LIN {X 0,Y 469.343,Z 366.999,A -85,B 0,C 180,E1 -7684.11,E2 -7684.11} C_VEL
LIN {X 0,Y 469.709,Z 359.682,A -85,B 0,C 180,E1 -7686.102,E2 -7686.102} C_VEL
LIN {X 0,Y 468.782,Z 353.417,A -85,B 0,C 180,E1 -7687.929,E2 -7687.929} C_VEL
LIN {X 0,Y 467.594,Z 347.243,A -85,B 0,C 180,E1 -7689.819,E2 -7689.819} C_VEL
LIN {X 0,Y 467.591,Z 347.243,A -85,B 0,C 180,E1 -7692.567,E2 -7692.567} C_VEL
LIN {X 0,Y 467.575,Z 347.246,A -85,B 0,C 180,E1 -7695.054,E2 -7695.054} C_VEL
LIN {X 0,Y 467.593,Z 347.241,A -85,B 0,C 180,E1 -7697.44,E2 -7697.44} C_VEL
LIN {X 0,Y 467.587,Z 347.243,A -85,B 0,C 180,E1 -7700.856,E2 -7700.856} C_VEL
LIN {X 0,Y 467.564,Z 347.245,A -85,B 0,C 180,E1 -7704.261,E2 -7704.261} C_VEL
LIN {X 0,Y 467.587,Z 347.242,A -85,B 0,C 180,E1 -7707.321,E2 -7707.321} C_VEL
LIN {X 0,Y 467.575,Z 347.245,A -85,B 0,C 180,E1 -7710.668,E2 -7710.668} C_VEL
LIN {X 0,Y 467.622,Z 347.237,A -85,B 0,C 180,E1 -7713.2,E2 -7713.2} C_VEL
LIN {X 0,Y 467.598,Z 347.242,A -85,B 0,C 180,E1 -7716.468,E2 -7716.468} C_VEL
LIN {X 0,Y 467.628,Z 347.236,A -85,B 0,C 180,E1 -7719.777,E2 -7719.777} C_VEL
LIN {X 0,Y 467.605,Z 347.24,A -85,B 0,C 180,E1 -7722.507,E2 -7722.507} C_VEL
LIN {X 0,Y 467.612,Z 347.238,A -85,B 0,C 180,E1 -7725.197,E2 -7725.197} C_VEL
LIN {X 0,Y 467.662,Z 347.233,A -85,B 0,C 180,E1 -7727.855,E2 -7727.855} C_VEL
LIN {X 0,Y 467.686,Z 347.227,A -85,B 0,C 180,E1 -7731.357,E2 -7731.357} C_VEL
LIN {X 0,Y 467.75,Z 347.221,A -85,B 0,C 180,E1 -7733.963,E2 -7733.963} C_VEL
LIN {X 0,Y 467.864,Z 347.206,A -85,B 0,C 180,E1 -7737.417,E2 -7737.417} C_VEL
LIN {X 0,Y 467.889,Z 347.206,A -85,B 0,C 180,E1 -7740,E2 -7740} C_VEL
LIN {X 0,Y 467.865,Z 347.207,A -85,B 0,C 180,E1 -7742.583,E2 -7742.583} C_VEL
LIN {X 0,Y 467.749,Z 347.222,A -85,B 0,C 180,E1 -7746.038,E2 -7746.038} C_VEL
LIN {X 0,Y 467.688,Z 347.229,A -85,B 0,C 180,E1 -7748.643,E2 -7748.643} C_VEL
LIN {X 0,Y 467.663,Z 347.235,A -85,B 0,C 180,E1 -7752.146,E2 -7752.146} C_VEL
LIN {X 0,Y 467.646,Z 347.236,A -85,B 0,C 180,E1 -7755.695,E2 -7755.695} C_VEL
LIN {X 0,Y 467.624,Z 347.236,A -85,B 0,C 180,E1 -7758.765,E2 -7758.765} C_VEL
LIN {X 0,Y 467.587,Z 347.242,A -85,B 0,C 180,E1 -7761.268,E2 -7761.268} C_VEL
LIN {X 0,Y 467.58,Z 347.243,A -85,B 0,C 180,E1 -7763.943,E2 -7763.943} C_VEL
LIN {X 0,Y 467.623,Z 347.236,A -85,B 0,C 180,E1 -7766.8,E2 -7766.8} C_VEL
LIN {X 0,Y 467.56,Z 347.246,A -85,B 0,C 180,E1 -7769.738,E2 -7769.738} C_VEL
LIN {X 0,Y 467.59,Z 347.241,A -85,B 0,C 180,E1 -7772.758,E2 -7772.758} C_VEL
LIN {X 0,Y 467.56,Z 347.245,A -85,B 0,C 180,E1 -7775.89,E2 -7775.89} C_VEL
LIN {X 0,Y 467.589,Z 347.242,A -85,B 0,C 180,E1 -7779.145,E2 -7779.145} C_VEL
LIN {X 0,Y 467.593,Z 347.24,A -85,B 0,C 180,E1 -7782.567,E2 -7782.567} C_VEL
LIN {X 0,Y 467.577,Z 347.244,A -85,B 0,C 180,E1 -7785.053,E2 -7785.053} C_VEL
LIN {X 0,Y 467.595,Z 347.241,A -85,B 0,C 180,E1 -7787.44,E2 -7787.44} C_VEL
LIN {X 0,Y 467.588,Z 347.242,A -85,B 0,C 180,E1 -7790.855,E2 -7790.855} C_VEL
LIN {X 0,Y 467.564,Z 347.243,A -85,B 0,C 180,E1 -7794.261,E2 -7794.261} C_VEL
LIN {X 0,Y 467.589,Z 347.242,A -85,B 0,C 180,E1 -7797.321,E2 -7797.321} C_VEL
LIN {X 0,Y 467.576,Z 347.245,A -85,B 0,C 180,E1 -7800.667,E2 -7800.667} C_VEL
LIN {X 0,Y 467.623,Z 347.238,A -85,B 0,C 180,E1 -7803.199,E2 -7803.199} C_VEL
LIN {X 0,Y 467.599,Z 347.241,A -85,B 0,C 180,E1 -7806.468,E2 -7806.468} C_VEL
LIN {X 0,Y 467.63,Z 347.235,A -85,B 0,C 180,E1 -7809.777,E2 -7809.777} C_VEL
LIN {X 0,Y 467.614,Z 347.239,A -85,B 0,C 180,E1 -7812.506,E2 -7812.506} C_VEL
LIN {X 0,Y 467.604,Z 347.238,A -85,B 0,C 180,E1 -7815.421,E2 -7815.421} C_VEL
LIN {X 0,Y 466.933,Z 347.324,A -85,B 0,C 180,E1 -7816.14,E2 -7816.14} C_VEL
LIN {X 0,Y 464.09,Z 347.677,A -85,B 0,C 180,E1 -7817.309,E2 -7817.309} C_VEL
LIN {X 0,Y 461.692,Z 347.976,A -85,B 0,C 180,E1 -7818.251,E2 -7818.251} C_VEL
LIN {X 0,Y 460.666,Z 348.105,A -85,B 0,C 180,E1 -7818.978,E2 -7818.978} C_VEL
LIN {X 0,Y 460.584,Z 348.115,A -85,B 0,C 180,E1 -7819.225,E2 -7819.225} C_VEL
LIN {X 0,Y 460.675,Z 348.104,A -85,B 0,C 180,E1 -7822.587,E2 -7822.587} C_VEL
LIN {X 0,Y 460.674,Z 348.304,A -85,B 0,C 180,E1 -7822.926,E2 -7822.926} C_VEL
LIN {X 0,Y 463.587,Z 358.571,A -85,B 0,C 180,E1 -7823.471,E2 -7823.471} C_VEL
LIN {X 0,Y 463.267,Z 370.178,A -85,B 0,C 180,E1 -7824.122,E2 -7824.122} C_VEL
LIN {X 0,Y 462.868,Z 380.748,A -85,B 0,C 180,E1 -7824.882,E2 -7824.882} C_VEL
LIN {X 0,Y 462.353,Z 391.565,A -85,B 0,C 180,E1 -7825.859,E2 -7825.859} C_VEL
LIN {X 0,Y 461.872,Z 401.21,A -85,B 0,C 180,E1 -7826.947,E2 -7826.947} C_VEL
LIN {X 0,Y 461.389,Z 410.564,A -85,B 0,C 180,E1 -7828.254,E2 -7828.254} C_VEL
LIN {X 0,Y 460.955,Z 418.019,A -85,B 0,C 180,E1 -7829.563,E2 -7829.563} C_VEL
LIN {X 0,Y 460.616,Z 424.017,A -85,B 0,C 180,E1 -7830.874,E2 -7830.874} C_VEL
LIN {X 0,Y 460.424,Z 428.772,A -85,B 0,C 180,E1 -7832.186,E2 -7832.186} C_VEL
LIN {X 0,Y 460.216,Z 432.455,A -85,B 0,C 180,E1 -7833.501,E2 -7833.501} C_VEL
LIN {X 0,Y 460.141,Z 434.354,A -85,B 0,C 180,E1 -7834.379,E2 -7834.379} C_VEL
LIN {X 0,Y 460.106,Z 435.844,A -85,B 0,C 180,E1 -7835.258,E2 -7835.258} C_VEL
LIN {X 0,Y 460.098,Z 437.555,A -85,B 0,C 180,E1 -7837.018,E2 -7837.018} C_VEL
LIN {X 0,Y 460.068,Z 437.759,A -85,B 0,C 180,E1 -7838.786,E2 -7838.786} C_VEL
LIN {X 0,Y 460.068,Z 436.331,A -85,B 0,C 180,E1 -7840.562,E2 -7840.562} C_VEL
LIN {X 0,Y 460.31,Z 433.443,A -85,B 0,C 180,E1 -7842.27,E2 -7842.27} C_VEL
LIN {X 0,Y 460.472,Z 429.812,A -85,B 0,C 180,E1 -7843.684,E2 -7843.684} C_VEL
LIN {X 0,Y 460.719,Z 425.206,A -85,B 0,C 180,E1 -7845.029,E2 -7845.029} C_VEL
LIN {X 0,Y 461.101,Z 418.242,A -85,B 0,C 180,E1 -7846.596,E2 -7846.596} C_VEL
LIN {X 0,Y 461.515,Z 410.521,A -85,B 0,C 180,E1 -7847.96,E2 -7847.96} C_VEL
LIN {X 0,Y 462.079,Z 401.988,A -85,B 0,C 180,E1 -7849.162,E2 -7849.162} C_VEL
LIN {X 0,Y 462.433,Z 392.799,A -85,B 0,C 180,E1 -7850.227,E2 -7850.227} C_VEL
LIN {X 0,Y 462.997,Z 381.824,A -85,B 0,C 180,E1 -7851.247,E2 -7851.247} C_VEL
LIN {X 0,Y 463.474,Z 370.955,A -85,B 0,C 180,E1 -7852.042,E2 -7852.042} C_VEL
LIN {X 0,Y 463.827,Z 358.885,A -85,B 0,C 180,E1 -7852.728,E2 -7852.728} C_VEL
LIN {X 0,Y 460.571,Z 348.116,A -85,B 0,C 180,E1 -7853.333,E2 -7853.333} C_VEL
LIN {X 0,Y 460.566,Z 348.118,A -85,B 0,C 180,E1 -7856.264,E2 -7856.264} C_VEL
LIN {X 0,Y 460.542,Z 348.122,A -85,B 0,C 180,E1 -7859.23,E2 -7859.23} C_VEL
LIN {X 0,Y 460.533,Z 348.125,A -85,B 0,C 180,E1 -7862.283,E2 -7862.283} C_VEL
LIN {X 0,Y 460.511,Z 348.127,A -85,B 0,C 180,E1 -7865.445,E2 -7865.445} C_VEL
LIN {X 0,Y 460.545,Z 348.12,A -85,B 0,C 180,E1 -7868.897,E2 -7868.897} C_VEL
LIN {X 0,Y 460.524,Z 348.121,A -85,B 0,C 180,E1 -7872.18,E2 -7872.18} C_VEL
LIN {X 0,Y 460.517,Z 348.125,A -85,B 0,C 180,E1 -7875.411,E2 -7875.411} C_VEL
LIN {X 0,Y 460.535,Z 348.123,A -85,B 0,C 180,E1 -7878.396,E2 -7878.396} C_VEL
LIN {X 0,Y 460.546,Z 348.12,A -85,B 0,C 180,E1 -7881.268,E2 -7881.268} C_VEL
LIN {X 0,Y 460.513,Z 348.124,A -85,B 0,C 180,E1 -7884.554,E2 -7884.554} C_VEL
LIN {X 0,Y 460.531,Z 348.116,A -85,B 0,C 180,E1 -7887.715,E2 -7887.715} C_VEL
LIN {X 0,Y 460.546,Z 348.106,A -85,B 0,C 180,E1 -7890.769,E2 -7890.769} C_VEL
LIN {X 0,Y 460.566,Z 348.116,A -85,B 0,C 180,E1 -7893.735,E2 -7893.735} C_VEL
LIN {X 0,Y 460.544,Z 348.114,A -85,B 0,C 180,E1 -7896.623,E2 -7896.623} C_VEL
LIN {X 0,Y 460.55,Z 348.12,A -85,B 0,C 180,E1 -7899.452,E2 -7899.452} C_VEL
LIN {X 0,Y 460.557,Z 348.113,A -85,B 0,C 180,E1 -7902.23,E2 -7902.23} C_VEL
LIN {X 0,Y 460.565,Z 348.117,A -85,B 0,C 180,E1 -7904.965,E2 -7904.965} C_VEL
LIN {X 0,Y 460.628,Z 348.109,A -85,B 0,C 180,E1 -7907.666,E2 -7907.666} C_VEL
LIN {X 0,Y 460.627,Z 348.11,A -85,B 0,C 180,E1 -7911.224,E2 -7911.224} C_VEL
LIN {X 0,Y 460.707,Z 348.094,A -85,B 0,C 180,E1 -7913.87,E2 -7913.87} C_VEL
LIN {X 0,Y 460.823,Z 348.086,A -85,B 0,C 180,E1 -7917.377,E2 -7917.377} C_VEL
LIN {X 0,Y 460.851,Z 348.076,A -85,B 0,C 180,E1 -7920,E2 -7920} C_VEL
LIN {X 0,Y 460.822,Z 348.085,A -85,B 0,C 180,E1 -7922.622,E2 -7922.622} C_VEL
LIN {X 0,Y 460.707,Z 348.097,A -85,B 0,C 180,E1 -7926.13,E2 -7926.13} C_VEL
LIN {X 0,Y 460.625,Z 348.108,A -85,B 0,C 180,E1 -7928.776,E2 -7928.776} C_VEL
LIN {X 0,Y 460.609,Z 348.111,A -85,B 0,C 180,E1 -7932.445,E2 -7932.445} C_VEL
LIN {X 0,Y 460.596,Z 348.113,A -85,B 0,C 180,E1 -7935.998,E2 -7935.998} C_VEL
LIN {X 0,Y 460.567,Z 348.117,A -85,B 0,C 180,E1 -7938.902,E2 -7938.902} C_VEL
LIN {X 0,Y 460.512,Z 348.124,A -85,B 0,C 180,E1 -7941.486,E2 -7941.486} C_VEL
LIN {X 0,Y 460.539,Z 348.122,A -85,B 0,C 180,E1 -7944.332,E2 -7944.332} C_VEL
LIN {X 0,Y 460.581,Z 348.118,A -85,B 0,C 180,E1 -7947.243,E2 -7947.243} C_VEL
LIN {X 0,Y 460.524,Z 348.125,A -85,B 0,C 180,E1 -7950.239,E2 -7950.239} C_VEL
LIN {X 0,Y 460.526,Z 348.123,A -85,B 0,C 180,E1 -7953.325,E2 -7953.325} C_VEL
LIN {X 0,Y 460.478,Z 348.128,A -85,B 0,C 180,E1 -7956.529,E2 -7956.529} C_VEL
LIN {X 0,Y 460.576,Z 348.116,A -85,B 0,C 180,E1 -7959.858,E2 -7959.858} C_VEL
LIN {X 0,Y 460.54,Z 348.121,A -85,B 0,C 180,E1 -7962.905,E2 -7962.905} C_VEL
LIN {X 0,Y 460.522,Z 348.122,A -85,B 0,C 180,E1 -7965.829,E2 -7965.829} C_VEL
LIN {X 0,Y 460.58,Z 348.181,A -85,B 0,C 180,E1 -7969.1,E2 -7969.1} C_VEL
LIN {X 0,Y 462.373,Z 357.576,A -85,B 0,C 180,E1 -7972.222,E2 -7972.222} C_VEL
LIN {X 0,Y 463.135,Z 362.334,A -85,B 0,C 180,E1 -7973.715,E2 -7973.715} C_VEL
LIN {X 0,Y 462.404,Z 372.802,A -85,B 0,C 180,E1 -7976.714,E2 -7976.714} C_VEL
LIN {X 0,Y 461.796,Z 384.189,A -85,B 0,C 180,E1 -7979.854,E2 -7979.854} C_VEL
LIN {X 0,Y 461.342,Z 395.24,A -85,B 0,C 180,E1 -7982.806,E2 -7982.806} C_VEL
LIN {X 0,Y 460.89,Z 408.274,A -85,B 0,C 180,E1 -7986.195,E2 -7986.195} C_VEL
LIN {X 0,Y 460.507,Z 421.091,A -85,B 0,C 180,E1 -7989.451,E2 -7989.451} C_VEL
LIN {X 0,Y 460.222,Z 433.977,A -85,B 0,C 180,E1 -7992.676,E2 -7992.676} C_VEL
LIN {X 0,Y 460.077,Z 440.376,A -85,B 0,C 180,E1 -7994.267,E2 -7994.267} C_VEL
LIN {X 0,Y 461.609,Z 453.753,A -85,B 0,C 180,E1 -7994.647,E2 -7994.647} C_VEL
LIN {X 0,Y 462.611,Z 464.777,A -85,B 0,C 180,E1 -7995.09,E2 -7995.09} C_VEL
LIN {X 0,Y 462.569,Z 473.994,A -85,B 0,C 180,E1 -7995.538,E2 -7995.538} C_VEL
LIN {X 0,Y 461.951,Z 485.65,A -85,B 0,C 180,E1 -7996.249,E2 -7996.249} C_VEL
LIN {X 0,Y 461.413,Z 496.8,A -85,B 0,C 180,E1 -7997.114,E2 -7997.114} C_VEL
LIN {X 0,Y 460.933,Z 507.224,A -85,B 0,C 180,E1 -7998.122,E2 -7998.122} C_VEL
LIN {X 0,Y 460.519,Z 516.495,A -85,B 0,C 180,E1 -7999.226,E2 -7999.226} C_VEL
LIN {X 0,Y 460.149,Z 525.563,A -85,B 0,C 180,E1 -8000.551,E2 -8000.551} C_VEL
LIN {X 0,Y 459.994,Z 532.899,A -85,B 0,C 180,E1 -8001.876,E2 -8001.876} C_VEL
LIN {X 0,Y 459.849,Z 539.606,A -85,B 0,C 180,E1 -8003.421,E2 -8003.421} C_VEL
LIN {X 0,Y 459.776,Z 544.037,A -85,B 0,C 180,E1 -8004.738,E2 -8004.738} C_VEL
LIN {X 0,Y 459.874,Z 546.409,A -85,B 0,C 180,E1 -8005.618,E2 -8005.618} C_VEL
LIN {X 0,Y 459.902,Z 548.327,A -85,B 0,C 180,E1 -8006.496,E2 -8006.496} C_VEL
LIN {X 0,Y 459.824,Z 549.756,A -85,B 0,C 180,E1 -8007.373,E2 -8007.373} C_VEL
LIN {X 0,Y 459.793,Z 550.781,A -85,B 0,C 180,E1 -8008.249,E2 -8008.249} C_VEL
LIN {X 0,Y 459.781,Z 551.41,A -85,B 0,C 180,E1 -8009.125,E2 -8009.125} C_VEL
LIN {X 0,Y 459.791,Z 551.638,A -85,B 0,C 180,E1 -8010.001,E2 -8010.001} C_VEL
LIN {X 0,Y 459.78,Z 551.419,A -85,B 0,C 180,E1 -8010.876,E2 -8010.876} C_VEL
LIN {X 0,Y 459.791,Z 550.802,A -85,B 0,C 180,E1 -8011.752,E2 -8011.752} C_VEL
LIN {X 0,Y 459.822,Z 549.788,A -85,B 0,C 180,E1 -8012.629,E2 -8012.629} C_VEL
LIN {X 0,Y 459.901,Z 548.365,A -85,B 0,C 180,E1 -8013.505,E2 -8013.505} C_VEL
LIN {X 0,Y 459.796,Z 545.342,A -85,B 0,C 180,E1 -8014.823,E2 -8014.823} C_VEL
LIN {X 0,Y 459.852,Z 541.27,A -85,B 0,C 180,E1 -8016.142,E2 -8016.142} C_VEL
LIN {X 0,Y 459.903,Z 534.994,A -85,B 0,C 180,E1 -8017.685,E2 -8017.685} C_VEL
LIN {X 0,Y 460.063,Z 528.156,A -85,B 0,C 180,E1 -8019.009,E2 -8019.009} C_VEL
LIN {X 0,Y 460.351,Z 519.691,A -85,B 0,C 180,E1 -8020.334,E2 -8020.334} C_VEL
LIN {X 0,Y 460.733,Z 511.012,A -85,B 0,C 180,E1 -8021.438,E2 -8021.438} C_VEL
LIN {X 0,Y 461.294,Z 500.154,A -85,B 0,C 180,E1 -8022.555,E2 -8022.555} C_VEL
LIN {X 0,Y 461.744,Z 489.738,A -85,B 0,C 180,E1 -8023.422,E2 -8023.422} C_VEL
LIN {X 0,Y 462.269,Z 478.129,A -85,B 0,C 180,E1 -8024.191,E2 -8024.191} C_VEL
LIN {X 0,Y 462.688,Z 466.113,A -85,B 0,C 180,E1 -8024.796,E2 -8024.796} C_VEL
LIN {X 0,Y 461.575,Z 455.302,A -85,B 0,C 180,E1 -8025.238,E2 -8025.238} C_VEL
LIN {X 0,Y 460.236,Z 442.458,A -85,B 0,C 180,E1 -8025.603,E2 -8025.603} C_VEL
LIN {X 0,Y 460.089,Z 440.581,A -85,B 0,C 180,E1 -8025.673,E2 -8025.673} C_VEL
LIN {X 0,Y 460.318,Z 427.872,A -85,B 0,C 180,E1 -8028.809,E2 -8028.809} C_VEL
LIN {X 0,Y 460.642,Z 415.245,A -85,B 0,C 180,E1 -8031.951,E2 -8031.951} C_VEL
LIN {X 0,Y 460.945,Z 403.943,A -85,B 0,C 180,E1 -8034.791,E2 -8034.791} C_VEL
LIN {X 0,Y 461.426,Z 390.688,A -85,B 0,C 180,E1 -8038.175,E2 -8038.175} C_VEL
LIN {X 0,Y 461.872,Z 377.817,A -85,B 0,C 180,E1 -8041.557,E2 -8041.557} C_VEL
LIN {X 0,Y 462.61,Z 364.146,A -85,B 0,C 180,E1 -8045.261,E2 -8045.261} C_VEL
LIN {X 0,Y 462.699,Z 360.133,A -85,B 0,C 180,E1 -8046.387,E2 -8046.387} C_VEL
LIN {X 0,Y 461.183,Z 351.48,A -85,B 0,C 180,E1 -8048.996,E2 -8048.996} C_VEL
LIN {X 0,Y 460.571,Z 348.117,A -85,B 0,C 180,E1 -8050.064,E2 -8050.064} C_VEL
LIN {X 0,Y 460.513,Z 348.125,A -85,B 0,C 180,E1 -8053.375,E2 -8053.375} C_VEL
LIN {X 0,Y 460.504,Z 348.124,A -85,B 0,C 180,E1 -8056.625,E2 -8056.625} C_VEL
LIN {X 0,Y 460.546,Z 348.117,A -85,B 0,C 180,E1 -8059.731,E2 -8059.731} C_VEL
LIN {X 0,Y 460.504,Z 348.124,A -85,B 0,C 180,E1 -8062.524,E2 -8062.524} C_VEL
LIN {X 0,Y 460.551,Z 348.117,A -85,B 0,C 180,E1 -8065.624,E2 -8065.624} C_VEL
LIN {X 0,Y 460.542,Z 348.121,A -85,B 0,C 180,E1 -8068.745,E2 -8068.745} C_VEL
LIN {X 0,Y 460.586,Z 348.114,A -85,B 0,C 180,E1 -8072.254,E2 -8072.254} C_VEL
LIN {X 0,Y 460.564,Z 348.117,A -85,B 0,C 180,E1 -8074.706,E2 -8074.706} C_VEL
LIN {X 0,Y 460.517,Z 348.121,A -85,B 0,C 180,E1 -8077.572,E2 -8077.572} C_VEL
LIN {X 0,Y 460.573,Z 348.116,A -85,B 0,C 180,E1 -8080.385,E2 -8080.385} C_VEL
LIN {X 0,Y 460.606,Z 348.11,A -85,B 0,C 180,E1 -8084.003,E2 -8084.003} C_VEL
LIN {X 0,Y 460.615,Z 348.109,A -85,B 0,C 180,E1 -8087.666,E2 -8087.666} C_VEL
LIN {X 0,Y 460.633,Z 348.106,A -85,B 0,C 180,E1 -8091.224,E2 -8091.224} C_VEL
LIN {X 0,Y 460.716,Z 348.097,A -85,B 0,C 180,E1 -8093.87,E2 -8093.87} C_VEL
LIN {X 0,Y 460.804,Z 348.085,A -85,B 0,C 180,E1 -8097.378,E2 -8097.378} C_VEL
LIN {X 0,Y 460.86,Z 348.082,A -85,B 0,C 180,E1 -8100,E2 -8100} C_VEL
LIN {X 0,Y 460.806,Z 348.086,A -85,B 0,C 180,E1 -8102.623,E2 -8102.623} C_VEL
LIN {X 0,Y 460.715,Z 348.099,A -85,B 0,C 180,E1 -8106.13,E2 -8106.13} C_VEL
LIN {X 0,Y 460.635,Z 348.107,A -85,B 0,C 180,E1 -8108.776,E2 -8108.776} C_VEL
LIN {X 0,Y 460.62,Z 348.109,A -85,B 0,C 180,E1 -8112.445,E2 -8112.445} C_VEL
LIN {X 0,Y 460.607,Z 348.112,A -85,B 0,C 180,E1 -8115.998,E2 -8115.998} C_VEL
LIN {X 0,Y 460.577,Z 348.114,A -85,B 0,C 180,E1 -8118.902,E2 -8118.902} C_VEL
LIN {X 0,Y 460.522,Z 348.123,A -85,B 0,C 180,E1 -8121.486,E2 -8121.486} C_VEL
LIN {X 0,Y 460.549,Z 348.118,A -85,B 0,C 180,E1 -8124.332,E2 -8124.332} C_VEL
LIN {X 0,Y 460.579,Z 348.115,A -85,B 0,C 180,E1 -8127.244,E2 -8127.244} C_VEL
LIN {X 0,Y 460.517,Z 348.122,A -85,B 0,C 180,E1 -8130.24,E2 -8130.24} C_VEL
LIN {X 0,Y 460.536,Z 348.121,A -85,B 0,C 180,E1 -8133.325,E2 -8133.325} C_VEL
LIN {X 0,Y 460.483,Z 348.125,A -85,B 0,C 180,E1 -8136.529,E2 -8136.529} C_VEL
LIN {X 0,Y 460.539,Z 348.12,A -85,B 0,C 180,E1 -8139.862,E2 -8139.862} C_VEL
LIN {X 0,Y 460.52,Z 348.123,A -85,B 0,C 180,E1 -8142.9,E2 -8142.9} C_VEL
LIN {X 0,Y 460.518,Z 348.122,A -85,B 0,C 180,E1 -8145.83,E2 -8145.83} C_VEL
LIN {X 0,Y 460.538,Z 348.12,A -85,B 0,C 180,E1 -8148.989,E2 -8148.989} C_VEL
LIN {X 0,Y 460.532,Z 348.122,A -85,B 0,C 180,E1 -8151.267,E2 -8151.267} C_VEL
LIN {X 0,Y 460.515,Z 348.121,A -85,B 0,C 180,E1 -8154.554,E2 -8154.554} C_VEL
LIN {X 0,Y 460.538,Z 348.119,A -85,B 0,C 180,E1 -8157.715,E2 -8157.715} C_VEL
LIN {X 0,Y 460.546,Z 348.12,A -85,B 0,C 180,E1 -8160.769,E2 -8160.769} C_VEL
LIN {X 0,Y 460.57,Z 348.115,A -85,B 0,C 180,E1 -8163.734,E2 -8163.734} C_VEL
LIN {X 0,Y 460.553,Z 348.118,A -85,B 0,C 180,E1 -8166.624,E2 -8166.624} C_VEL
LIN {X 0,Y 460.558,Z 348.117,A -85,B 0,C 180,E1 -8169.452,E2 -8169.452} C_VEL
LIN {X 0,Y 460.565,Z 348.116,A -85,B 0,C 180,E1 -8172.23,E2 -8172.23} C_VEL
LIN {X 0,Y 460.572,Z 348.117,A -85,B 0,C 180,E1 -8174.964,E2 -8174.964} C_VEL
LIN {X 0,Y 460.618,Z 348.112,A -85,B 0,C 180,E1 -8178.559,E2 -8178.559} C_VEL
LIN {X 0,Y 460.584,Z 348.115,A -85,B 0,C 180,E1 -8179.225,E2 -8179.225} C_VEL
LIN {X 0,Y 459.911,Z 348.2,A -85,B 0,C 180,E1 -8179.712,E2 -8179.712} C_VEL
LIN {X 0,Y 457.082,Z 348.551,A -85,B 0,C 180,E1 -8180.473,E2 -8180.473} C_VEL
LIN {X 0,Y 454.253,Z 348.902,A -85,B 0,C 180,E1 -8181.244,E2 -8181.244} C_VEL
LIN {X 0,Y 453.601,Z 348.983,A -85,B 0,C 180,E1 -8181.741,E2 -8181.741} C_VEL
LIN {X 0,Y 453.663,Z 349.057,A -85,B 0,C 180,E1 -8182.707,E2 -8182.707} C_VEL
LIN {X 0,Y 456.713,Z 360.367,A -85,B 0,C 180,E1 -8183.317,E2 -8183.317} C_VEL
LIN {X 0,Y 456.34,Z 372.631,A -85,B 0,C 180,E1 -8184.032,E2 -8184.032} C_VEL
LIN {X 0,Y 455.825,Z 384.133,A -85,B 0,C 180,E1 -8184.913,E2 -8184.913} C_VEL
LIN {X 0,Y 455.386,Z 394.432,A -85,B 0,C 180,E1 -8185.906,E2 -8185.906} C_VEL
LIN {X 0,Y 454.881,Z 402.889,A -85,B 0,C 180,E1 -8186.9,E2 -8186.9} C_VEL
LIN {X 0,Y 454.472,Z 410.664,A -85,B 0,C 180,E1 -8188.005,E2 -8188.005} C_VEL
LIN {X 0,Y 454.014,Z 418.305,A -85,B 0,C 180,E1 -8189.334,E2 -8189.334} C_VEL
LIN {X 0,Y 453.583,Z 425.302,A -85,B 0,C 180,E1 -8190.887,E2 -8190.887} C_VEL
LIN {X 0,Y 453.404,Z 429.967,A -85,B 0,C 180,E1 -8192.22,E2 -8192.22} C_VEL
LIN {X 0,Y 453.17,Z 433.572,A -85,B 0,C 180,E1 -8193.556,E2 -8193.556} C_VEL
LIN {X 0,Y 453.11,Z 435.43,A -85,B 0,C 180,E1 -8194.447,E2 -8194.447} C_VEL
LIN {X 0,Y 453.073,Z 436.851,A -85,B 0,C 180,E1 -8195.34,E2 -8195.34} C_VEL
LIN {X 0,Y 453.061,Z 438.482,A -85,B 0,C 180,E1 -8197.128,E2 -8197.128} C_VEL
LIN {X 0,Y 453.057,Z 438.738,A -85,B 0,C 180,E1 -8198.025,E2 -8198.025} C_VEL
LIN {X 0,Y 453.028,Z 438.582,A -85,B 0,C 180,E1 -8198.924,E2 -8198.924} C_VEL
LIN {X 0,Y 453.049,Z 437.075,A -85,B 0,C 180,E1 -8200.728,E2 -8200.728} C_VEL
LIN {X 0,Y 453.299,Z 434.276,A -85,B 0,C 180,E1 -8202.374,E2 -8202.374} C_VEL
LIN {X 0,Y 453.483,Z 430.357,A -85,B 0,C 180,E1 -8203.899,E2 -8203.899} C_VEL
LIN {X 0,Y 453.781,Z 425.66,A -85,B 0,C 180,E1 -8205.265,E2 -8205.265} C_VEL
LIN {X 0,Y 454.115,Z 419.893,A -85,B 0,C 180,E1 -8206.59,E2 -8206.59} C_VEL
LIN {X 0,Y 454.56,Z 412.156,A -85,B 0,C 180,E1 -8208.012,E2 -8208.012} C_VEL
LIN {X 0,Y 455.161,Z 403.549,A -85,B 0,C 180,E1 -8209.267,E2 -8209.267} C_VEL
LIN {X 0,Y 455.586,Z 393.763,A -85,B 0,C 180,E1 -8210.427,E2 -8210.427} C_VEL
LIN {X 0,Y 456.179,Z 382.816,A -85,B 0,C 180,E1 -8211.462,E2 -8211.462} C_VEL
LIN {X 0,Y 456.744,Z 370.74,A -85,B 0,C 180,E1 -8212.348,E2 -8212.348} C_VEL
LIN {X 0,Y 457.008,Z 360.188,A -85,B 0,C 180,E1 -8212.955,E2 -8212.955} C_VEL
LIN {X 0,Y 453.505,Z 348.996,A -85,B 0,C 180,E1 -8213.607,E2 -8213.607} C_VEL
LIN {X 0,Y 453.509,Z 348.998,A -85,B 0,C 180,E1 -8216.705,E2 -8216.705} C_VEL
LIN {X 0,Y 453.474,Z 349.004,A -85,B 0,C 180,E1 -8219.784,E2 -8219.784} C_VEL
LIN {X 0,Y 453.492,Z 349,A -85,B 0,C 180,E1 -8223.188,E2 -8223.188} C_VEL
LIN {X 0,Y 453.454,Z 349.004,A -85,B 0,C 180,E1 -8226.298,E2 -8226.298} C_VEL
LIN {X 0,Y 453.505,Z 348.997,A -85,B 0,C 180,E1 -8229.447,E2 -8229.447} C_VEL
LIN {X 0,Y 453.468,Z 349.001,A -85,B 0,C 180,E1 -8232.993,E2 -8232.993} C_VEL
LIN {X 0,Y 453.466,Z 349.002,A -85,B 0,C 180,E1 -8235.778,E2 -8235.778} C_VEL
LIN {X 0,Y 453.515,Z 348.997,A -85,B 0,C 180,E1 -8239.405,E2 -8239.405} C_VEL
LIN {X 0,Y 453.477,Z 349.001,A -85,B 0,C 180,E1 -8242.222,E2 -8242.222} C_VEL
LIN {X 0,Y 453.488,Z 348.999,A -85,B 0,C 180,E1 -8245.222,E2 -8245.222} C_VEL
LIN {X 0,Y 453.467,Z 348.991,A -85,B 0,C 180,E1 -8248.474,E2 -8248.474} C_VEL
LIN {X 0,Y 453.514,Z 348.983,A -85,B 0,C 180,E1 -8251.288,E2 -8251.288} C_VEL
LIN {X 0,Y 453.523,Z 348.994,A -85,B 0,C 180,E1 -8254.284,E2 -8254.284} C_VEL
LIN {X 0,Y 453.477,Z 348.994,A -85,B 0,C 180,E1 -8257.204,E2 -8257.204} C_VEL
LIN {X 0,Y 453.503,Z 348.996,A -85,B 0,C 180,E1 -8260.066,E2 -8260.066} C_VEL
LIN {X 0,Y 453.505,Z 348.992,A -85,B 0,C 180,E1 -8262.875,E2 -8262.875} C_VEL
LIN {X 0,Y 453.513,Z 348.995,A -85,B 0,C 180,E1 -8265.644,E2 -8265.644} C_VEL
LIN {X 0,Y 453.579,Z 348.988,A -85,B 0,C 180,E1 -8268.379,E2 -8268.379} C_VEL
LIN {X 0,Y 453.649,Z 348.978,A -85,B 0,C 180,E1 -8271.985,E2 -8271.985} C_VEL
LIN {X 0,Y 453.669,Z 348.97,A -85,B 0,C 180,E1 -8274.666,E2 -8274.666} C_VEL
LIN {X 0,Y 453.763,Z 348.965,A -85,B 0,C 180,E1 -8277.337,E2 -8277.337} C_VEL
LIN {X 0,Y 453.821,Z 348.951,A -85,B 0,C 180,E1 -8280,E2 -8280} C_VEL
LIN {X 0,Y 453.763,Z 348.964,A -85,B 0,C 180,E1 -8282.663,E2 -8282.663} C_VEL
LIN {X 0,Y 453.674,Z 348.974,A -85,B 0,C 180,E1 -8286.225,E2 -8286.225} C_VEL
LIN {X 0,Y 453.589,Z 348.984,A -85,B 0,C 180,E1 -8288.913,E2 -8288.913} C_VEL
LIN {X 0,Y 453.559,Z 348.989,A -85,B 0,C 180,E1 -8292.529,E2 -8292.529} C_VEL
LIN {X 0,Y 453.541,Z 348.993,A -85,B 0,C 180,E1 -8296.196,E2 -8296.196} C_VEL
LIN {X 0,Y 453.517,Z 348.995,A -85,B 0,C 180,E1 -8299.041,E2 -8299.041} C_VEL
LIN {X 0,Y 453.473,Z 349.001,A -85,B 0,C 180,E1 -8301.836,E2 -8301.836} C_VEL
LIN {X 0,Y 453.511,Z 348.997,A -85,B 0,C 180,E1 -8304.735,E2 -8304.735} C_VEL
LIN {X 0,Y 453.535,Z 348.995,A -85,B 0,C 180,E1 -8307.962,E2 -8307.962} C_VEL
LIN {X 0,Y 453.48,Z 349.001,A -85,B 0,C 180,E1 -8310.759,E2 -8310.759} C_VEL
LIN {X 0,Y 453.475,Z 349.001,A -85,B 0,C 180,E1 -8313.913,E2 -8313.913} C_VEL
LIN {X 0,Y 453.47,Z 349.001,A -85,B 0,C 180,E1 -8317.188,E2 -8317.188} C_VEL
LIN {X 0,Y 453.531,Z 348.992,A -85,B 0,C 180,E1 -8319.446,E2 -8319.446} C_VEL
LIN {X 0,Y 453.49,Z 349,A -85,B 0,C 180,E1 -8322.992,E2 -8322.992} C_VEL
LIN {X 0,Y 453.475,Z 349,A -85,B 0,C 180,E1 -8325.781,E2 -8325.781} C_VEL
LIN {X 0,Y 453.537,Z 349.105,A -85,B 0,C 180,E1 -8328.773,E2 -8328.773} C_VEL
LIN {X 0,Y 455.266,Z 358.195,A -85,B 0,C 180,E1 -8331.868,E2 -8331.868} C_VEL
LIN {X 0,Y 456.179,Z 363.971,A -85,B 0,C 180,E1 -8333.717,E2 -8333.717} C_VEL
LIN {X 0,Y 455.378,Z 374.801,A -85,B 0,C 180,E1 -8336.865,E2 -8336.865} C_VEL
LIN {X 0,Y 454.763,Z 385.741,A -85,B 0,C 180,E1 -8339.933,E2 -8339.933} C_VEL
LIN {X 0,Y 454.23,Z 398.309,A -85,B 0,C 180,E1 -8343.341,E2 -8343.341} C_VEL
LIN {X 0,Y 453.747,Z 411.179,A -85,B 0,C 180,E1 -8346.737,E2 -8346.737} C_VEL
LIN {X 0,Y 453.369,Z 424.046,A -85,B 0,C 180,E1 -8350.061,E2 -8350.061} C_VEL
LIN {X 0,Y 453.07,Z 436.846,A -85,B 0,C 180,E1 -8353.324,E2 -8353.324} C_VEL
LIN {X 0,Y 453.006,Z 439.653,A -85,B 0,C 180,E1 -8353.995,E2 -8353.995} C_VEL
LIN {X 0,Y 454.599,Z 452.76,A -85,B 0,C 180,E1 -8354.38,E2 -8354.38} C_VEL
LIN {X 0,Y 455.54,Z 464.34,A -85,B 0,C 180,E1 -8354.853,E2 -8354.853} C_VEL
LIN {X 0,Y 455.825,Z 469.154,A -85,B 0,C 180,E1 -8355.091,E2 -8355.091} C_VEL
LIN {X 0,Y 455.179,Z 481.81,A -85,B 0,C 180,E1 -8355.812,E2 -8355.812} C_VEL
LIN {X 0,Y 454.648,Z 492.379,A -85,B 0,C 180,E1 -8356.593,E2 -8356.593} C_VEL
LIN {X 0,Y 454.179,Z 503.293,A -85,B 0,C 180,E1 -8357.603,E2 -8357.603} C_VEL
LIN {X 0,Y 453.663,Z 512.229,A -85,B 0,C 180,E1 -8358.609,E2 -8358.609} C_VEL
LIN {X 0,Y 453.175,Z 521.985,A -85,B 0,C 180,E1 -8359.953,E2 -8359.953} C_VEL
LIN {X 0,Y 452.946,Z 529.789,A -85,B 0,C 180,E1 -8361.299,E2 -8361.299} C_VEL
LIN {X 0,Y 452.82,Z 535.161,A -85,B 0,C 180,E1 -8362.42,E2 -8362.42} C_VEL
LIN {X 0,Y 452.78,Z 540.383,A -85,B 0,C 180,E1 -8363.763,E2 -8363.763} C_VEL
LIN {X 0,Y 452.729,Z 544.444,A -85,B 0,C 180,E1 -8365.103,E2 -8365.103} C_VEL
LIN {X 0,Y 452.858,Z 547.47,A -85,B 0,C 180,E1 -8366.442,E2 -8366.442} C_VEL
LIN {X 0,Y 452.741,Z 549.916,A -85,B 0,C 180,E1 -8368.222,E2 -8368.222} C_VEL
LIN {X 0,Y 452.732,Z 550.542,A -85,B 0,C 180,E1 -8369.111,E2 -8369.111} C_VEL
LIN {X 0,Y 452.745,Z 550.765,A -85,B 0,C 180,E1 -8370.001,E2 -8370.001} C_VEL
LIN {X 0,Y 452.732,Z 550.542,A -85,B 0,C 180,E1 -8370.89,E2 -8370.89} C_VEL
LIN {X 0,Y 452.741,Z 549.921,A -85,B 0,C 180,E1 -8371.78,E2 -8371.78} C_VEL
LIN {X 0,Y 452.77,Z 548.904,A -85,B 0,C 180,E1 -8372.67,E2 -8372.67} C_VEL
LIN {X 0,Y 452.856,Z 547.475,A -85,B 0,C 180,E1 -8373.56,E2 -8373.56} C_VEL
LIN {X 0,Y 452.734,Z 544.44,A -85,B 0,C 180,E1 -8374.898,E2 -8374.898} C_VEL
LIN {X 0,Y 452.781,Z 540.354,A -85,B 0,C 180,E1 -8376.238,E2 -8376.238} C_VEL
LIN {X 0,Y 452.852,Z 534.059,A -85,B 0,C 180,E1 -8377.805,E2 -8377.805} C_VEL
LIN {X 0,Y 453.014,Z 527.202,A -85,B 0,C 180,E1 -8379.15,E2 -8379.15} C_VEL
LIN {X 0,Y 453.316,Z 518.712,A -85,B 0,C 180,E1 -8380.497,E2 -8380.497} C_VEL
LIN {X 0,Y 453.705,Z 509.991,A -85,B 0,C 180,E1 -8381.618,E2 -8381.618} C_VEL
LIN {X 0,Y 454.244,Z 500.234,A -85,B 0,C 180,E1 -8382.645,E2 -8382.645} C_VEL
LIN {X 0,Y 454.71,Z 490.083,A -85,B 0,C 180,E1 -8383.52,E2 -8383.52} C_VEL
LIN {X 0,Y 455.247,Z 478.771,A -85,B 0,C 180,E1 -8384.301,E2 -8384.301} C_VEL
LIN {X 0,Y 455.708,Z 467.338,A -85,B 0,C 180,E1 -8384.914,E2 -8384.914} C_VEL
LIN {X 0,Y 454.508,Z 454.047,A -85,B 0,C 180,E1 -8385.471,E2 -8385.471} C_VEL
LIN {X 0,Y 452.99,Z 439.797,A -85,B 0,C 180,E1 -8385.88,E2 -8385.88} C_VEL
LIN {X 0,Y 453.252,Z 427.396,A -85,B 0,C 180,E1 -8389.004,E2 -8389.004} C_VEL
LIN {X 0,Y 453.606,Z 414.364,A -85,B 0,C 180,E1 -8392.309,E2 -8392.309} C_VEL
LIN {X 0,Y 453.926,Z 403.084,A -85,B 0,C 180,E1 -8395.2,E2 -8395.2} C_VEL
LIN {X 0,Y 454.399,Z 391.694,A -85,B 0,C 180,E1 -8398.164,E2 -8398.164} C_VEL
LIN {X 0,Y 454.913,Z 378.016,A -85,B 0,C 180,E1 -8401.821,E2 -8401.821} C_VEL
LIN {X 0,Y 455.665,Z 364.804,A -85,B 0,C 180,E1 -8405.466,E2 -8405.466} C_VEL
LIN {X 0,Y 455.624,Z 360.631,A -85,B 0,C 180,E1 -8406.669,E2 -8406.669} C_VEL
LIN {X 0,Y 454.052,Z 351.796,A -85,B 0,C 180,E1 -8409.392,E2 -8409.392} C_VEL
LIN {X 0,Y 453.506,Z 348.998,A -85,B 0,C 180,E1 -8410.307,E2 -8410.307} C_VEL
LIN {X 0,Y 453.468,Z 349.003,A -85,B 0,C 180,E1 -8413.246,E2 -8413.246} C_VEL
LIN {X 0,Y 453.471,Z 349.001,A -85,B 0,C 180,E1 -8415.779,E2 -8415.779} C_VEL
LIN {X 0,Y 453.483,Z 348.997,A -85,B 0,C 180,E1 -8418.21,E2 -8418.21} C_VEL
LIN {X 0,Y 453.515,Z 348.997,A -85,B 0,C 180,E1 -8420.791,E2 -8420.791} C_VEL
LIN {X 0,Y 453.459,Z 349,A -85,B 0,C 180,E1 -8423.918,E2 -8423.918} C_VEL
LIN {X 0,Y 453.488,Z 349,A -85,B 0,C 180,E1 -8427.152,E2 -8427.152} C_VEL
LIN {X 0,Y 453.48,Z 348.998,A -85,B 0,C 180,E1 -8430.269,E2 -8430.269} C_VEL
LIN {X 0,Y 453.512,Z 348.994,A -85,B 0,C 180,E1 -8433.294,E2 -8433.294} C_VEL
LIN {X 0,Y 453.509,Z 348.995,A -85,B 0,C 180,E1 -8436.239,E2 -8436.239} C_VEL
LIN {X 0,Y 453.488,Z 348.998,A -85,B 0,C 180,E1 -8439.118,E2 -8439.118} C_VEL
LIN {X 0,Y 453.51,Z 348.994,A -85,B 0,C 180,E1 -8441.945,E2 -8441.945} C_VEL
LIN {X 0,Y 453.545,Z 348.991,A -85,B 0,C 180,E1 -8444.727,E2 -8444.727} C_VEL
LIN {X 0,Y 453.565,Z 348.989,A -85,B 0,C 180,E1 -8448.379,E2 -8448.379} C_VEL
LIN {X 0,Y 453.658,Z 348.977,A -85,B 0,C 180,E1 -8451.985,E2 -8451.985} C_VEL
LIN {X 0,Y 453.676,Z 348.975,A -85,B 0,C 180,E1 -8454.667,E2 -8454.667} C_VEL
LIN {X 0,Y 453.749,Z 348.963,A -85,B 0,C 180,E1 -8457.337,E2 -8457.337} C_VEL
LIN {X 0,Y 453.83,Z 348.957,A -85,B 0,C 180,E1 -8460,E2 -8460} C_VEL
LIN {X 0,Y 453.75,Z 348.965,A -85,B 0,C 180,E1 -8462.663,E2 -8462.663} C_VEL
LIN {X 0,Y 453.683,Z 348.975,A -85,B 0,C 180,E1 -8466.225,E2 -8466.225} C_VEL
LIN {X 0,Y 453.599,Z 348.983,A -85,B 0,C 180,E1 -8468.913,E2 -8468.913} C_VEL
LIN {X 0,Y 453.57,Z 348.987,A -85,B 0,C 180,E1 -8472.529,E2 -8472.529} C_VEL
LIN {X 0,Y 453.551,Z 348.991,A -85,B 0,C 180,E1 -8476.196,E2 -8476.196} C_VEL
LIN {X 0,Y 453.527,Z 348.992,A -85,B 0,C 180,E1 -8479.041,E2 -8479.041} C_VEL
LIN {X 0,Y 453.483,Z 348.999,A -85,B 0,C 180,E1 -8481.836,E2 -8481.836} C_VEL
LIN {X 0,Y 453.521,Z 348.992,A -85,B 0,C 180,E1 -8484.734,E2 -8484.734} C_VEL
LIN {X 0,Y 453.538,Z 348.992,A -85,B 0,C 180,E1 -8487.96,E2 -8487.96} C_VEL
LIN {X 0,Y 453.473,Z 349.001,A -85,B 0,C 180,E1 -8491.525,E2 -8491.525} C_VEL
LIN {X 0,Y 453.494,Z 348.996,A -85,B 0,C 180,E1 -8494.777,E2 -8494.777} C_VEL
LIN {X 0,Y 453.471,Z 348.998,A -85,B 0,C 180,E1 -8498.311,E2 -8498.311} C_VEL
LIN {X 0,Y 453.5,Z 348.995,A -85,B 0,C 180,E1 -8500.609,E2 -8500.609} C_VEL
LIN {X 0,Y 453.462,Z 349.002,A -85,B 0,C 180,E1 -8503.244,E2 -8503.244} C_VEL
LIN {X 0,Y 453.473,Z 349,A -85,B 0,C 180,E1 -8505.779,E2 -8505.779} C_VEL
LIN {X 0,Y 453.486,Z 348.997,A -85,B 0,C 180,E1 -8508.209,E2 -8508.209} C_VEL
LIN {X 0,Y 453.5,Z 348.997,A -85,B 0,C 180,E1 -8510.793,E2 -8510.793} C_VEL
LIN {X 0,Y 453.458,Z 349,A -85,B 0,C 180,E1 -8513.917,E2 -8513.917} C_VEL
LIN {X 0,Y 453.49,Z 349,A -85,B 0,C 180,E1 -8517.151,E2 -8517.151} C_VEL
LIN {X 0,Y 453.481,Z 348.997,A -85,B 0,C 180,E1 -8520.268,E2 -8520.268} C_VEL
LIN {X 0,Y 453.513,Z 348.995,A -85,B 0,C 180,E1 -8523.294,E2 -8523.294} C_VEL
LIN {X 0,Y 453.51,Z 348.995,A -85,B 0,C 180,E1 -8526.238,E2 -8526.238} C_VEL
LIN {X 0,Y 453.49,Z 348.999,A -85,B 0,C 180,E1 -8529.117,E2 -8529.117} C_VEL
LIN {X 0,Y 453.517,Z 348.993,A -85,B 0,C 180,E1 -8531.944,E2 -8531.944} C_VEL
LIN {X 0,Y 453.547,Z 348.992,A -85,B 0,C 180,E1 -8534.726,E2 -8534.726} C_VEL
LIN {X 0,Y 453.567,Z 348.989,A -85,B 0,C 180,E1 -8538.379,E2 -8538.379} C_VEL
LIN {X 0,Y 453.601,Z 348.983,A -85,B 0,C 180,E1 -8541.741,E2 -8541.741} C_VEL
LIN {X 0,Y 453.491,Z 349.648,A -85,B 0,C 180,E1 -8542.089,E2 -8542.089} C_VEL
LIN {X 0,Y 453.082,Z 351.905,A -85,B 0,C 180,E1 -8542.481,E2 -8542.481} C_VEL
LIN {X 0,Y 452.314,Z 356.003,A -85,B 0,C 180,E1 -8542.862,E2 -8542.862} C_VEL
LIN {X 0,Y 451.259,Z 361.724,A -85,B 0,C 180,E1 -8543.189,E2 -8543.189} C_VEL
LIN {X 0,Y 449.645,Z 371.587,A -85,B 0,C 180,E1 -8543.713,E2 -8543.713} C_VEL
LIN {X 0,Y 449.404,Z 375.159,A -85,B 0,C 180,E1 -8543.958,E2 -8543.958} C_VEL
LIN {X 0,Y 448.87,Z 386.141,A -85,B 0,C 180,E1 -8544.834,E2 -8544.834} C_VEL
LIN {X 0,Y 448.396,Z 396.251,A -85,B 0,C 180,E1 -8545.842,E2 -8545.842} C_VEL
LIN {X 0,Y 447.906,Z 404.543,A -85,B 0,C 180,E1 -8546.851,E2 -8546.851} C_VEL
LIN {X 0,Y 447.397,Z 413.524,A -85,B 0,C 180,E1 -8548.199,E2 -8548.199} C_VEL
LIN {X 0,Y 446.912,Z 420.765,A -85,B 0,C 180,E1 -8549.549,E2 -8549.549} C_VEL
LIN {X 0,Y 446.553,Z 426.576,A -85,B 0,C 180,E1 -8550.901,E2 -8550.901} C_VEL
LIN {X 0,Y 446.38,Z 431.154,A -85,B 0,C 180,E1 -8552.255,E2 -8552.255} C_VEL
LIN {X 0,Y 446.124,Z 434.683,A -85,B 0,C 180,E1 -8553.612,E2 -8553.612} C_VEL
LIN {X 0,Y 446.079,Z 436.491,A -85,B 0,C 180,E1 -8554.518,E2 -8554.518} C_VEL
LIN {X 0,Y 446.005,Z 438.819,A -85,B 0,C 180,E1 -8556.332,E2 -8556.332} C_VEL
LIN {X 0,Y 446.026,Z 439.409,A -85,B 0,C 180,E1 -8557.241,E2 -8557.241} C_VEL
LIN {X 0,Y 446.004,Z 439.618,A -85,B 0,C 180,E1 -8558.152,E2 -8558.152} C_VEL
LIN {X 0,Y 445.987,Z 438.806,A -85,B 0,C 180,E1 -8559.981,E2 -8559.981} C_VEL
LIN {X 0,Y 446.034,Z 437.823,A -85,B 0,C 180,E1 -8560.898,E2 -8560.898} C_VEL
LIN {X 0,Y 446.285,Z 435.121,A -85,B 0,C 180,E1 -8562.48,E2 -8562.48} C_VEL
LIN {X 0,Y 446.52,Z 430.909,A -85,B 0,C 180,E1 -8564.12,E2 -8564.12} C_VEL
LIN {X 0,Y 446.846,Z 426.126,A -85,B 0,C 180,E1 -8565.507,E2 -8565.507} C_VEL
LIN {X 0,Y 447.224,Z 420.264,A -85,B 0,C 180,E1 -8566.853,E2 -8566.853} C_VEL
LIN {X 0,Y 447.725,Z 412.399,A -85,B 0,C 180,E1 -8568.296,E2 -8568.296} C_VEL
LIN {X 0,Y 448.32,Z 403.97,A -85,B 0,C 180,E1 -8569.526,E2 -8569.526} C_VEL
LIN {X 0,Y 448.852,Z 393.673,A -85,B 0,C 180,E1 -8570.747,E2 -8570.747} C_VEL
LIN {X 0,Y 449.371,Z 383.839,A -85,B 0,C 180,E1 -8571.683,E2 -8571.683} C_VEL
LIN {X 0,Y 449.964,Z 372.682,A -85,B 0,C 180,E1 -8572.524,E2 -8572.524} C_VEL
LIN {X 0,Y 450.31,Z 362.249,A -85,B 0,C 180,E1 -8573.147,E2 -8573.147} C_VEL
LIN {X 0,Y 446.482,Z 349.87,A -85,B 0,C 180,E1 -8573.903,E2 -8573.903} C_VEL
LIN {X 0,Y 446.477,Z 349.873,A -85,B 0,C 180,E1 -8577.16,E2 -8577.16} C_VEL
LIN {X 0,Y 446.429,Z 349.882,A -85,B 0,C 180,E1 -8580.249,E2 -8580.249} C_VEL
LIN {X 0,Y 446.446,Z 349.876,A -85,B 0,C 180,E1 -8583.453,E2 -8583.453} C_VEL
LIN {X 0,Y 446.402,Z 349.883,A -85,B 0,C 180,E1 -8586.744,E2 -8586.744} C_VEL
LIN {X 0,Y 446.469,Z 349.873,A -85,B 0,C 180,E1 -8589.526,E2 -8589.526} C_VEL
LIN {X 0,Y 446.432,Z 349.879,A -85,B 0,C 180,E1 -8592.603,E2 -8592.603} C_VEL
LIN {X 0,Y 446.454,Z 349.875,A -85,B 0,C 180,E1 -8595.102,E2 -8595.102} C_VEL
LIN {X 0,Y 446.435,Z 349.879,A -85,B 0,C 180,E1 -8598.609,E2 -8598.609} C_VEL
LIN {X 0,Y 446.475,Z 349.872,A -85,B 0,C 180,E1 -8600.976,E2 -8600.976} C_VEL
LIN {X 0,Y 446.42,Z 349.878,A -85,B 0,C 180,E1 -8604.374,E2 -8604.374} C_VEL
LIN {X 0,Y 446.427,Z 349.873,A -85,B 0,C 180,E1 -8607.638,E2 -8607.638} C_VEL
LIN {X 0,Y 446.468,Z 349.858,A -85,B 0,C 180,E1 -8610.792,E2 -8610.792} C_VEL
LIN {X 0,Y 446.475,Z 349.87,A -85,B 0,C 180,E1 -8613.848,E2 -8613.848} C_VEL
LIN {X 0,Y 446.427,Z 349.871,A -85,B 0,C 180,E1 -8616.823,E2 -8616.823} C_VEL
LIN {X 0,Y 446.442,Z 349.875,A -85,B 0,C 180,E1 -8619.737,E2 -8619.737} C_VEL
LIN {X 0,Y 446.461,Z 349.869,A -85,B 0,C 180,E1 -8622.597,E2 -8622.597} C_VEL
LIN {X 0,Y 446.47,Z 349.874,A -85,B 0,C 180,E1 -8625.412,E2 -8625.412} C_VEL
LIN {X 0,Y 446.539,Z 349.865,A -85,B 0,C 180,E1 -8628.193,E2 -8628.193} C_VEL
LIN {X 0,Y 446.597,Z 349.856,A -85,B 0,C 180,E1 -8631.858,E2 -8631.858} C_VEL
LIN {X 0,Y 446.644,Z 349.845,A -85,B 0,C 180,E1 -8634.582,E2 -8634.582} C_VEL
LIN {X 0,Y 446.707,Z 349.844,A -85,B 0,C 180,E1 -8637.294,E2 -8637.294} C_VEL
LIN {X 0,Y 446.792,Z 349.826,A -85,B 0,C 180,E1 -8640,E2 -8640} C_VEL
LIN {X 0,Y 446.706,Z 349.843,A -85,B 0,C 180,E1 -8642.705,E2 -8642.705} C_VEL
LIN {X 0,Y 446.644,Z 349.85,A -85,B 0,C 180,E1 -8646.324,E2 -8646.324} C_VEL
LIN {X 0,Y 446.535,Z 349.863,A -85,B 0,C 180,E1 -8649.055,E2 -8649.055} C_VEL
LIN {X 0,Y 446.517,Z 349.865,A -85,B 0,C 180,E1 -8652.73,E2 -8652.73} C_VEL
LIN {X 0,Y 446.492,Z 349.871,A -85,B 0,C 180,E1 -8656.228,E2 -8656.228} C_VEL
LIN {X 0,Y 446.466,Z 349.874,A -85,B 0,C 180,E1 -8659.303,E2 -8659.303} C_VEL
LIN {X 0,Y 446.415,Z 349.882,A -85,B 0,C 180,E1 -8662.2,E2 -8662.2} C_VEL
LIN {X 0,Y 446.455,Z 349.877,A -85,B 0,C 180,E1 -8665.152,E2 -8665.152} C_VEL
LIN {X 0,Y 446.48,Z 349.874,A -85,B 0,C 180,E1 -8668.179,E2 -8668.179} C_VEL
LIN {X 0,Y 446.417,Z 349.881,A -85,B 0,C 180,E1 -8671.3,E2 -8671.3} C_VEL
LIN {X 0,Y 446.428,Z 349.878,A -85,B 0,C 180,E1 -8674.523,E2 -8674.523} C_VEL
LIN {X 0,Y 446.437,Z 349.871,A -85,B 0,C 180,E1 -8678.084,E2 -8678.084} C_VEL
LIN {X 0,Y 446.444,Z 349.874,A -85,B 0,C 180,E1 -8680.921,E2 -8680.921} C_VEL
LIN {X 0,Y 446.443,Z 349.873,A -85,B 0,C 180,E1 -8683.841,E2 -8683.841} C_VEL
LIN {X 0,Y 446.445,Z 349.871,A -85,B 0,C 180,E1 -8686.397,E2 -8686.397} C_VEL
LIN {X 0,Y 446.483,Z 349.984,A -85,B 0,C 180,E1 -8688.428,E2 -8688.428} C_VEL
LIN {X 0,Y 447.975,Z 357.731,A -85,B 0,C 180,E1 -8691.132,E2 -8691.132} C_VEL
LIN {X 0,Y 449.215,Z 364.977,A -85,B 0,C 180,E1 -8693.523,E2 -8693.523} C_VEL
LIN {X 0,Y 448.578,Z 373.746,A -85,B 0,C 180,E1 -8696.137,E2 -8696.137} C_VEL
LIN {X 0,Y 447.896,Z 384.745,A -85,B 0,C 180,E1 -8699.3,E2 -8699.3} C_VEL
LIN {X 0,Y 447.341,Z 395.855,A -85,B 0,C 180,E1 -8702.39,E2 -8702.39} C_VEL
LIN {X 0,Y 446.823,Z 408.676,A -85,B 0,C 180,E1 -8705.862,E2 -8705.862} C_VEL
LIN {X 0,Y 446.392,Z 421.481,A -85,B 0,C 180,E1 -8709.254,E2 -8709.254} C_VEL
LIN {X 0,Y 446.057,Z 434.248,A -85,B 0,C 180,E1 -8712.581,E2 -8712.581} C_VEL
LIN {X 0,Y 445.938,Z 438.758,A -85,B 0,C 180,E1 -8713.707,E2 -8713.707} C_VEL
LIN {X 0,Y 447.603,Z 451.903,A -85,B 0,C 180,E1 -8714.105,E2 -8714.105} C_VEL
LIN {X 0,Y 448.649,Z 465.278,A -85,B 0,C 180,E1 -8714.673,E2 -8714.673} C_VEL
LIN {X 0,Y 448.856,Z 470.957,A -85,B 0,C 180,E1 -8714.97,E2 -8714.97} C_VEL
LIN {X 0,Y 448.167,Z 482.854,A -85,B 0,C 180,E1 -8715.701,E2 -8715.701} C_VEL
LIN {X 0,Y 447.515,Z 494.78,A -85,B 0,C 180,E1 -8716.646,E2 -8716.646} C_VEL
LIN {X 0,Y 447.064,Z 504.761,A -85,B 0,C 180,E1 -8717.633,E2 -8717.633} C_VEL
LIN {X 0,Y 446.555,Z 513.301,A -85,B 0,C 180,E1 -8718.655,E2 -8718.655} C_VEL
LIN {X 0,Y 446.047,Z 522.599,A -85,B 0,C 180,E1 -8720.02,E2 -8720.02} C_VEL
LIN {X 0,Y 445.857,Z 530.136,A -85,B 0,C 180,E1 -8721.388,E2 -8721.388} C_VEL
LIN {X 0,Y 445.693,Z 536.203,A -85,B 0,C 180,E1 -8722.754,E2 -8722.754} C_VEL
LIN {X 0,Y 445.727,Z 541.026,A -85,B 0,C 180,E1 -8724.118,E2 -8724.118} C_VEL
LIN {X 0,Y 445.736,Z 544.713,A -85,B 0,C 180,E1 -8725.479,E2 -8725.479} C_VEL
LIN {X 0,Y 445.797,Z 546.619,A -85,B 0,C 180,E1 -8726.385,E2 -8726.385} C_VEL
LIN {X 0,Y 445.688,Z 549.054,A -85,B 0,C 180,E1 -8728.193,E2 -8728.193} C_VEL
LIN {X 0,Y 445.683,Z 549.677,A -85,B 0,C 180,E1 -8729.097,E2 -8729.097} C_VEL
LIN {X 0,Y 445.699,Z 549.892,A -85,B 0,C 180,E1 -8730.001,E2 -8730.001} C_VEL
LIN {X 0,Y 445.685,Z 549.662,A -85,B 0,C 180,E1 -8730.904,E2 -8730.904} C_VEL
LIN {X 0,Y 445.691,Z 549.036,A -85,B 0,C 180,E1 -8731.808,E2 -8731.808} C_VEL
LIN {X 0,Y 445.72,Z 548.013,A -85,B 0,C 180,E1 -8732.712,E2 -8732.712} C_VEL
LIN {X 0,Y 445.812,Z 546.575,A -85,B 0,C 180,E1 -8733.616,E2 -8733.616} C_VEL
LIN {X 0,Y 445.676,Z 543.527,A -85,B 0,C 180,E1 -8734.976,E2 -8734.976} C_VEL
LIN {X 0,Y 445.709,Z 538.518,A -85,B 0,C 180,E1 -8736.588,E2 -8736.588} C_VEL
LIN {X 0,Y 445.832,Z 532.072,A -85,B 0,C 180,E1 -8738.157,E2 -8738.157} C_VEL
LIN {X 0,Y 445.984,Z 524.952,A -85,B 0,C 180,E1 -8739.525,E2 -8739.525} C_VEL
LIN {X 0,Y 446.361,Z 516.052,A -85,B 0,C 180,E1 -8740.892,E2 -8740.892} C_VEL
LIN {X 0,Y 446.889,Z 505.964,A -85,B 0,C 180,E1 -8742.143,E2 -8742.143} C_VEL
LIN {X 0,Y 447.336,Z 496.025,A -85,B 0,C 180,E1 -8743.142,E2 -8743.142} C_VEL
LIN {X 0,Y 447.985,Z 484.384,A -85,B 0,C 180,E1 -8744.074,E2 -8744.074} C_VEL
LIN {X 0,Y 448.598,Z 471.668,A -85,B 0,C 180,E1 -8744.866,E2 -8744.866} C_VEL
LIN {X 0,Y 448.543,Z 465.958,A -85,B 0,C 180,E1 -8745.158,E2 -8745.158} C_VEL
LIN {X 0,Y 447.391,Z 452.877,A -85,B 0,C 180,E1 -8745.707,E2 -8745.707} C_VEL
LIN {X 0,Y 445.908,Z 438.991,A -85,B 0,C 180,E1 -8746.106,E2 -8746.106} C_VEL
LIN {X 0,Y 446.174,Z 427.422,A -85,B 0,C 180,E1 -8749.073,E2 -8749.073} C_VEL
LIN {X 0,Y 446.519,Z 415.333,A -85,B 0,C 180,E1 -8752.195,E2 -8752.195} C_VEL
LIN {X 0,Y 446.842,Z 404.085,A -85,B 0,C 180,E1 -8755.13,E2 -8755.13} C_VEL
LIN {X 0,Y 447.391,Z 391.781,A -85,B 0,C 180,E1 -8758.394,E2 -8758.394} C_VEL
LIN {X 0,Y 447.849,Z 379.842,A -85,B 0,C 180,E1 -8761.64,E2 -8761.64} C_VEL
LIN {X 0,Y 448.495,Z 368.234,A -85,B 0,C 180,E1 -8764.888,E2 -8764.888} C_VEL
LIN {X 0,Y 448.794,Z 364.466,A -85,B 0,C 180,E1 -8765.962,E2 -8765.962} C_VEL
LIN {X 0,Y 448.361,Z 360.082,A -85,B 0,C 180,E1 -8767.28,E2 -8767.28} C_VEL
LIN {X 0,Y 446.477,Z 349.873,A -85,B 0,C 180,E1 -8770.533,E2 -8770.533} C_VEL
LIN {X 0,Y 446.427,Z 349.881,A -85,B 0,C 180,E1 -8773.844,E2 -8773.844} C_VEL
LIN {X 0,Y 446.404,Z 349.882,A -85,B 0,C 180,E1 -8776.404,E2 -8776.404} C_VEL
LIN {X 0,Y 446.431,Z 349.878,A -85,B 0,C 180,E1 -8779.083,E2 -8779.083} C_VEL
LIN {X 0,Y 446.42,Z 349.877,A -85,B 0,C 180,E1 -8781.921,E2 -8781.921} C_VEL
LIN {X 0,Y 446.433,Z 349.876,A -85,B 0,C 180,E1 -8785.477,E2 -8785.477} C_VEL
LIN {X 0,Y 446.422,Z 349.88,A -85,B 0,C 180,E1 -8788.7,E2 -8788.7} C_VEL
LIN {X 0,Y 446.489,Z 349.868,A -85,B 0,C 180,E1 -8791.822,E2 -8791.822} C_VEL
LIN {X 0,Y 446.463,Z 349.874,A -85,B 0,C 180,E1 -8794.848,E2 -8794.848} C_VEL
LIN {X 0,Y 446.454,Z 349.874,A -85,B 0,C 180,E1 -8798.245,E2 -8798.245} C_VEL
LIN {X 0,Y 446.458,Z 349.872,A -85,B 0,C 180,E1 -8801.649,E2 -8801.649} C_VEL
LIN {X 0,Y 446.513,Z 349.868,A -85,B 0,C 180,E1 -8804.48,E2 -8804.48} C_VEL
LIN {X 0,Y 446.523,Z 349.866,A -85,B 0,C 180,E1 -8808.193,E2 -8808.193} C_VEL
LIN {X 0,Y 446.606,Z 349.854,A -85,B 0,C 180,E1 -8811.858,E2 -8811.858} C_VEL
LIN {X 0,Y 446.651,Z 349.85,A -85,B 0,C 180,E1 -8814.583,E2 -8814.583} C_VEL
LIN {X 0,Y 446.67,Z 349.848,A -85,B 0,C 180,E1 -8818.197,E2 -8818.197} C_VEL
LIN {X 0,Y 446.8,Z 349.832,A -85,B 0,C 180,E1 -8820,E2 -8820} C_VEL
LIN {X 0,Y 446.697,Z 349.844,A -85,B 0,C 180,E1 -8822.706,E2 -8822.706} C_VEL
LIN {X 0,Y 446.652,Z 349.851,A -85,B 0,C 180,E1 -8826.324,E2 -8826.324} C_VEL
LIN {X 0,Y 446.545,Z 349.861,A -85,B 0,C 180,E1 -8829.055,E2 -8829.055} C_VEL
LIN {X 0,Y 446.528,Z 349.863,A -85,B 0,C 180,E1 -8832.73,E2 -8832.73} C_VEL
LIN {X 0,Y 446.503,Z 349.869,A -85,B 0,C 180,E1 -8836.228,E2 -8836.228} C_VEL
LIN {X 0,Y 446.476,Z 349.871,A -85,B 0,C 180,E1 -8839.303,E2 -8839.303} C_VEL
LIN {X 0,Y 446.425,Z 349.878,A -85,B 0,C 180,E1 -8842.2,E2 -8842.2} C_VEL
LIN {X 0,Y 446.464,Z 349.872,A -85,B 0,C 180,E1 -8845.152,E2 -8845.152} C_VEL
LIN {X 0,Y 446.491,Z 349.869,A -85,B 0,C 180,E1 -8848.179,E2 -8848.179} C_VEL
LIN {X 0,Y 446.426,Z 349.878,A -85,B 0,C 180,E1 -8851.775,E2 -8851.775} C_VEL
LIN {X 0,Y 446.435,Z 349.875,A -85,B 0,C 180,E1 -8854.523,E2 -8854.523} C_VEL
LIN {X 0,Y 446.422,Z 349.877,A -85,B 0,C 180,E1 -8858.079,E2 -8858.079} C_VEL
LIN {X 0,Y 446.433,Z 349.876,A -85,B 0,C 180,E1 -8860.918,E2 -8860.918} C_VEL
LIN {X 0,Y 446.408,Z 349.879,A -85,B 0,C 180,E1 -8863.846,E2 -8863.846} C_VEL
LIN {X 0,Y 446.406,Z 349.878,A -85,B 0,C 180,E1 -8866.403,E2 -8866.403} C_VEL
LIN {X 0,Y 446.434,Z 349.878,A -85,B 0,C 180,E1 -8869.082,E2 -8869.082} C_VEL
LIN {X 0,Y 446.414,Z 349.877,A -85,B 0,C 180,E1 -8872.121,E2 -8872.121} C_VEL
LIN {X 0,Y 446.435,Z 349.877,A -85,B 0,C 180,E1 -8875.477,E2 -8875.477} C_VEL
LIN {X 0,Y 446.423,Z 349.879,A -85,B 0,C 180,E1 -8878.699,E2 -8878.699} C_VEL
LIN {X 0,Y 446.491,Z 349.867,A -85,B 0,C 180,E1 -8881.821,E2 -8881.821} C_VEL
LIN {X 0,Y 446.465,Z 349.874,A -85,B 0,C 180,E1 -8884.847,E2 -8884.847} C_VEL
LIN {X 0,Y 446.455,Z 349.873,A -85,B 0,C 180,E1 -8888.245,E2 -8888.245} C_VEL
LIN {X 0,Y 446.463,Z 349.872,A -85,B 0,C 180,E1 -8891.649,E2 -8891.649} C_VEL
LIN {X 0,Y 446.514,Z 349.867,A -85,B 0,C 180,E1 -8894.479,E2 -8894.479} C_VEL
LIN {X 0,Y 446.525,Z 349.864,A -85,B 0,C 180,E1 -8898.193,E2 -8898.193} C_VEL
LIN {X 0,Y 446.572,Z 349.86,A -85,B 0,C 180,E1 -8901.751,E2 -8901.751} C_VEL
LIN {X 0,Y 446.605,Z 349.873,A -85,B 0,C 180,E1 -8902.484,E2 -8902.484} C_VEL
LIN {X 0,Y 449.773,Z 361.05,A -85,B 0,C 180,E1 -8903.1,E2 -8903.1} C_VEL
LIN {X 0,Y 449.468,Z 373.335,A -85,B 0,C 180,E1 -8903.828,E2 -8903.828} C_VEL
LIN {X 0,Y 449.404,Z 375.159,A -85,B 0,C 180,E1 -8903.958,E2 -8903.958} C_VEL
LIN {X 0,Y 448.647,Z 380.342,A -85,B 0,C 180,E1 -8904.325,E2 -8904.325} C_VEL
LIN {X 0,Y 445.506,Z 388.517,A -85,B 0,C 180,E1 -8904.926,E2 -8904.926} C_VEL
LIN {X 0,Y 442.23,Z 396.228,A -85,B 0,C 180,E1 -8905.605,E2 -8905.605} C_VEL
LIN {X 0,Y 441.266,Z 400.628,A -85,B 0,C 180,E1 -8906.089,E2 -8906.089} C_VEL
LIN {X 0,Y 440.738,Z 409.326,A -85,B 0,C 180,E1 -8907.257,E2 -8907.257} C_VEL
LIN {X 0,Y 440.285,Z 417.523,A -85,B 0,C 180,E1 -8908.627,E2 -8908.627} C_VEL
LIN {X 0,Y 439.808,Z 424.146,A -85,B 0,C 180,E1 -8909.999,E2 -8909.999} C_VEL
LIN {X 0,Y 439.47,Z 429.438,A -85,B 0,C 180,E1 -8911.374,E2 -8911.374} C_VEL
LIN {X 0,Y 439.244,Z 433.578,A -85,B 0,C 180,E1 -8912.751,E2 -8912.751} C_VEL
LIN {X 0,Y 439.08,Z 435.788,A -85,B 0,C 180,E1 -8913.67,E2 -8913.67} C_VEL
LIN {X 0,Y 439.05,Z 437.523,A -85,B 0,C 180,E1 -8914.59,E2 -8914.59} C_VEL
LIN {X 0,Y 438.965,Z 439.779,A -85,B 0,C 180,E1 -8916.434,E2 -8916.434} C_VEL
LIN {X 0,Y 438.976,Z 440.336,A -85,B 0,C 180,E1 -8917.358,E2 -8917.358} C_VEL
LIN {X 0,Y 438.964,Z 440.475,A -85,B 0,C 180,E1 -8918.284,E2 -8918.284} C_VEL
LIN {X 0,Y 438.977,Z 439.591,A -85,B 0,C 180,E1 -8920.143,E2 -8920.143} C_VEL
LIN {X 0,Y 439.024,Z 438.57,A -85,B 0,C 180,E1 -8921.075,E2 -8921.075} C_VEL
LIN {X 0,Y 439.293,Z 435.943,A -85,B 0,C 180,E1 -8922.601,E2 -8922.601} C_VEL
LIN {X 0,Y 439.56,Z 431.471,A -85,B 0,C 180,E1 -8924.348,E2 -8924.348} C_VEL
LIN {X 0,Y 439.913,Z 426.603,A -85,B 0,C 180,E1 -8925.758,E2 -8925.758} C_VEL
LIN {X 0,Y 440.358,Z 420.425,A -85,B 0,C 180,E1 -8927.172,E2 -8927.172} C_VEL
LIN {X 0,Y 440.9,Z 412.619,A -85,B 0,C 180,E1 -8928.59,E2 -8928.59} C_VEL
LIN {X 0,Y 441.568,Z 403.141,A -85,B 0,C 180,E1 -8929.961,E2 -8929.961} C_VEL
LIN {X 0,Y 442.084,Z 393.589,A -85,B 0,C 180,E1 -8931.08,E2 -8931.08} C_VEL
LIN {X 0,Y 442.668,Z 383.473,A -85,B 0,C 180,E1 -8932.029,E2 -8932.029} C_VEL
LIN {X 0,Y 443.269,Z 371.409,A -85,B 0,C 180,E1 -8932.923,E2 -8932.923} C_VEL
LIN {X 0,Y 443.503,Z 363.531,A -85,B 0,C 180,E1 -8933.393,E2 -8933.393} C_VEL
LIN {X 0,Y 439.728,Z 352.02,A -85,B 0,C 180,E1 -8934.119,E2 -8934.119} C_VEL
LIN {X 0,Y 439.444,Z 350.747,A -85,B 0,C 180,E1 -8934.201,E2 -8934.201} C_VEL
LIN {X 0,Y 439.443,Z 350.751,A -85,B 0,C 180,E1 -8937.632,E2 -8937.632} C_VEL
LIN {X 0,Y 439.363,Z 350.758,A -85,B 0,C 180,E1 -8940.788,E2 -8940.788} C_VEL
LIN {X 0,Y 439.388,Z 350.753,A -85,B 0,C 180,E1 -8944.043,E2 -8944.043} C_VEL
LIN {X 0,Y 439.349,Z 350.761,A -85,B 0,C 180,E1 -8946.886,E2 -8946.886} C_VEL
LIN {X 0,Y 439.406,Z 350.751,A -85,B 0,C 180,E1 -8949.849,E2 -8949.849} C_VEL
LIN {X 0,Y 439.385,Z 350.756,A -85,B 0,C 180,E1 -8952.627,E2 -8952.627} C_VEL
LIN {X 0,Y 439.402,Z 350.754,A -85,B 0,C 180,E1 -8955.27,E2 -8955.27} C_VEL
LIN {X 0,Y 439.397,Z 350.755,A -85,B 0,C 180,E1 -8958.741,E2 -8958.741} C_VEL
LIN {X 0,Y 439.392,Z 350.756,A -85,B 0,C 180,E1 -8961.604,E2 -8961.604} C_VEL
LIN {X 0,Y 439.4,Z 350.753,A -85,B 0,C 180,E1 -8964.844,E2 -8964.844} C_VEL
LIN {X 0,Y 439.385,Z 350.747,A -85,B 0,C 180,E1 -8968.14,E2 -8968.14} C_VEL
LIN {X 0,Y 439.423,Z 350.738,A -85,B 0,C 180,E1 -8971.327,E2 -8971.327} C_VEL
LIN {X 0,Y 439.403,Z 350.753,A -85,B 0,C 180,E1 -8974.415,E2 -8974.415} C_VEL
LIN {X 0,Y 439.363,Z 350.753,A -85,B 0,C 180,E1 -8977.424,E2 -8977.424} C_VEL
LIN {X 0,Y 439.439,Z 350.747,A -85,B 0,C 180,E1 -8980.662,E2 -8980.662} C_VEL
LIN {X 0,Y 439.46,Z 350.745,A -85,B 0,C 180,E1 -8984.224,E2 -8984.224} C_VEL
LIN {X 0,Y 439.506,Z 350.74,A -85,B 0,C 180,E1 -8988.002,E2 -8988.002} C_VEL
LIN {X 0,Y 439.545,Z 350.735,A -85,B 0,C 180,E1 -8991.726,E2 -8991.726} C_VEL
LIN {X 0,Y 439.619,Z 350.719,A -85,B 0,C 180,E1 -8994.496,E2 -8994.496} C_VEL
LIN {X 0,Y 439.633,Z 350.725,A -85,B 0,C 180,E1 -8998.168,E2 -8998.168} C_VEL
LIN {X 0,Y 439.762,Z 350.702,A -85,B 0,C 180,E1 -9000,E2 -9000} C_VEL
LIN {X 0,Y 439.653,Z 350.722,A -85,B 0,C 180,E1 -9002.749,E2 -9002.749} C_VEL
LIN {X 0,Y 439.615,Z 350.726,A -85,B 0,C 180,E1 -9006.425,E2 -9006.425} C_VEL
LIN {X 0,Y 439.496,Z 350.738,A -85,B 0,C 180,E1 -9009.202,E2 -9009.202} C_VEL
LIN {X 0,Y 439.461,Z 350.744,A -85,B 0,C 180,E1 -9012.938,E2 -9012.938} C_VEL
LIN {X 0,Y 439.443,Z 350.748,A -85,B 0,C 180,E1 -9016.349,E2 -9016.349} C_VEL
LIN {X 0,Y 439.399,Z 350.753,A -85,B 0,C 180,E1 -9019.626,E2 -9019.626} C_VEL
LIN {X 0,Y 439.362,Z 350.759,A -85,B 0,C 180,E1 -9022.576,E2 -9022.576} C_VEL
LIN {X 0,Y 439.402,Z 350.754,A -85,B 0,C 180,E1 -9025.585,E2 -9025.585} C_VEL
LIN {X 0,Y 439.421,Z 350.752,A -85,B 0,C 180,E1 -9028.673,E2 -9028.673} C_VEL
LIN {X 0,Y 439.371,Z 350.758,A -85,B 0,C 180,E1 -9031.861,E2 -9031.861} C_VEL
LIN {X 0,Y 439.398,Z 350.754,A -85,B 0,C 180,E1 -9035.156,E2 -9035.156} C_VEL
LIN {X 0,Y 439.397,Z 350.746,A -85,B 0,C 180,E1 -9038.594,E2 -9038.594} C_VEL
LIN {X 0,Y 439.402,Z 350.747,A -85,B 0,C 180,E1 -9041.26,E2 -9041.26} C_VEL
LIN {X 0,Y 439.408,Z 350.749,A -85,B 0,C 180,E1 -9044.728,E2 -9044.728} C_VEL
LIN {X 0,Y 439.441,Z 350.795,A -85,B 0,C 180,E1 -9048.045,E2 -9048.045} C_VEL
LIN {X 0,Y 440.992,Z 358.789,A -85,B 0,C 180,E1 -9050.903,E2 -9050.903} C_VEL
LIN {X 0,Y 442.276,Z 366.279,A -85,B 0,C 180,E1 -9053.424,E2 -9053.424} C_VEL
LIN {X 0,Y 441.586,Z 375.265,A -85,B 0,C 180,E1 -9056.15,E2 -9056.15} C_VEL
LIN {X 0,Y 440.864,Z 386.421,A -85,B 0,C 180,E1 -9059.411,E2 -9059.411} C_VEL
LIN {X 0,Y 440.298,Z 397.068,A -85,B 0,C 180,E1 -9062.427,E2 -9062.427} C_VEL
LIN {X 0,Y 439.766,Z 408.681,A -85,B 0,C 180,E1 -9065.634,E2 -9065.634} C_VEL
LIN {X 0,Y 439.357,Z 420.777,A -85,B 0,C 180,E1 -9068.906,E2 -9068.906} C_VEL
LIN {X 0,Y 438.979,Z 433.468,A -85,B 0,C 180,E1 -9072.291,E2 -9072.291} C_VEL
LIN {X 0,Y 438.883,Z 437.621,A -85,B 0,C 180,E1 -9073.39,E2 -9073.39} C_VEL
LIN {X 0,Y 440.723,Z 452.081,A -85,B 0,C 180,E1 -9073.856,E2 -9073.856} C_VEL
LIN {X 0,Y 441.622,Z 464.923,A -85,B 0,C 180,E1 -9074.423,E2 -9074.423} C_VEL
LIN {X 0,Y 441.961,Z 470.523,A -85,B 0,C 180,E1 -9074.73,E2 -9074.73} C_VEL
LIN {X 0,Y 441.261,Z 482.317,A -85,B 0,C 180,E1 -9075.473,E2 -9075.473} C_VEL
LIN {X 0,Y 440.612,Z 493.467,A -85,B 0,C 180,E1 -9076.369,E2 -9076.369} C_VEL
LIN {X 0,Y 440.105,Z 504.09,A -85,B 0,C 180,E1 -9077.434,E2 -9077.434} C_VEL
LIN {X 0,Y 439.538,Z 512.585,A -85,B 0,C 180,E1 -9078.471,E2 -9078.471} C_VEL
LIN {X 0,Y 439.005,Z 521.843,A -85,B 0,C 180,E1 -9079.858,E2 -9079.858} C_VEL
LIN {X 0,Y 438.784,Z 529.353,A -85,B 0,C 180,E1 -9081.248,E2 -9081.248} C_VEL
LIN {X 0,Y 438.621,Z 535.4,A -85,B 0,C 180,E1 -9082.636,E2 -9082.636} C_VEL
LIN {X 0,Y 438.641,Z 540.204,A -85,B 0,C 180,E1 -9084.023,E2 -9084.023} C_VEL
LIN {X 0,Y 438.641,Z 543.875,A -85,B 0,C 180,E1 -9085.406,E2 -9085.406} C_VEL
LIN {X 0,Y 438.722,Z 545.77,A -85,B 0,C 180,E1 -9086.327,E2 -9086.327} C_VEL
LIN {X 0,Y 438.667,Z 547.184,A -85,B 0,C 180,E1 -9087.246,E2 -9087.246} C_VEL
LIN {X 0,Y 438.635,Z 548.196,A -85,B 0,C 180,E1 -9088.164,E2 -9088.164} C_VEL
LIN {X 0,Y 438.633,Z 548.814,A -85,B 0,C 180,E1 -9089.083,E2 -9089.083} C_VEL
LIN {X 0,Y 438.653,Z 549.017,A -85,B 0,C 180,E1 -9090.001,E2 -9090.001} C_VEL
LIN {X 0,Y 438.637,Z 548.78,A -85,B 0,C 180,E1 -9090.919,E2 -9090.919} C_VEL
LIN {X 0,Y 438.642,Z 548.148,A -85,B 0,C 180,E1 -9091.837,E2 -9091.837} C_VEL
LIN {X 0,Y 438.669,Z 547.118,A -85,B 0,C 180,E1 -9092.756,E2 -9092.756} C_VEL
LIN {X 0,Y 438.769,Z 545.667,A -85,B 0,C 180,E1 -9093.674,E2 -9093.674} C_VEL
LIN {X 0,Y 438.6,Z 542.601,A -85,B 0,C 180,E1 -9095.057,E2 -9095.057} C_VEL
LIN {X 0,Y 438.645,Z 537.907,A -85,B 0,C 180,E1 -9096.601,E2 -9096.601} C_VEL
LIN {X 0,Y 438.759,Z 531.099,A -85,B 0,C 180,E1 -9098.289,E2 -9098.289} C_VEL
LIN {X 0,Y 438.923,Z 523.946,A -85,B 0,C 180,E1 -9099.679,E2 -9099.679} C_VEL
LIN {X 0,Y 439.332,Z 515.01,A -85,B 0,C 180,E1 -9101.068,E2 -9101.068} C_VEL
LIN {X 0,Y 439.927,Z 504.89,A -85,B 0,C 180,E1 -9102.338,E2 -9102.338} C_VEL
LIN {X 0,Y 440.397,Z 494.354,A -85,B 0,C 180,E1 -9103.4,E2 -9103.4} C_VEL
LIN {X 0,Y 440.998,Z 483.158,A -85,B 0,C 180,E1 -9104.302,E2 -9104.302} C_VEL
LIN {X 0,Y 441.646,Z 471.362,A -85,B 0,C 180,E1 -9105.046,E2 -9105.046} C_VEL
LIN {X 0,Y 441.405,Z 465.693,A -85,B 0,C 180,E1 -9105.35,E2 -9105.35} C_VEL
LIN {X 0,Y 440.333,Z 452.469,A -85,B 0,C 180,E1 -9105.922,E2 -9105.922} C_VEL
LIN {X 0,Y 438.844,Z 438.048,A -85,B 0,C 180,E1 -9106.366,E2 -9106.366} C_VEL
LIN {X 0,Y 439.134,Z 425.536,A -85,B 0,C 180,E1 -9109.639,E2 -9109.639} C_VEL
LIN {X 0,Y 439.462,Z 414.424,A -85,B 0,C 180,E1 -9112.571,E2 -9112.571} C_VEL
LIN {X 0,Y 439.847,Z 403.203,A -85,B 0,C 180,E1 -9115.558,E2 -9115.558} C_VEL
LIN {X 0,Y 440.372,Z 391.873,A -85,B 0,C 180,E1 -9118.627,E2 -9118.627} C_VEL
LIN {X 0,Y 440.892,Z 379.529,A -85,B 0,C 180,E1 -9122.051,E2 -9122.051} C_VEL
LIN {X 0,Y 441.636,Z 367.928,A -85,B 0,C 180,E1 -9125.364,E2 -9125.364} C_VEL
LIN {X 0,Y 441.719,Z 363.64,A -85,B 0,C 180,E1 -9126.631,E2 -9126.631} C_VEL
LIN {X 0,Y 440.398,Z 355.858,A -85,B 0,C 180,E1 -9129.097,E2 -9129.097} C_VEL
LIN {X 0,Y 439.431,Z 350.752,A -85,B 0,C 180,E1 -9130.837,E2 -9130.837} C_VEL
LIN {X 0,Y 439.389,Z 350.757,A -85,B 0,C 180,E1 -9133.964,E2 -9133.964} C_VEL
LIN {X 0,Y 439.356,Z 350.759,A -85,B 0,C 180,E1 -9136.541,E2 -9136.541} C_VEL
LIN {X 0,Y 439.385,Z 350.756,A -85,B 0,C 180,E1 -9139.02,E2 -9139.02} C_VEL
LIN {X 0,Y 439.381,Z 350.754,A -85,B 0,C 180,E1 -9141.608,E2 -9141.608} C_VEL
LIN {X 0,Y 439.404,Z 350.753,A -85,B 0,C 180,E1 -9144.844,E2 -9144.844} C_VEL
LIN {X 0,Y 439.379,Z 350.753,A -85,B 0,C 180,E1 -9148.14,E2 -9148.14} C_VEL
LIN {X 0,Y 439.437,Z 350.747,A -85,B 0,C 180,E1 -9151.598,E2 -9151.598} C_VEL
LIN {X 0,Y 439.411,Z 350.753,A -85,B 0,C 180,E1 -9154.416,E2 -9154.416} C_VEL
LIN {X 0,Y 439.371,Z 350.755,A -85,B 0,C 180,E1 -9157.425,E2 -9157.425} C_VEL
LIN {X 0,Y 439.446,Z 350.749,A -85,B 0,C 180,E1 -9160.663,E2 -9160.663} C_VEL
LIN {X 0,Y 439.468,Z 350.745,A -85,B 0,C 180,E1 -9164.225,E2 -9164.225} C_VEL
LIN {X 0,Y 439.489,Z 350.742,A -85,B 0,C 180,E1 -9168.002,E2 -9168.002} C_VEL
LIN {X 0,Y 439.554,Z 350.732,A -85,B 0,C 180,E1 -9171.727,E2 -9171.727} C_VEL
LIN {X 0,Y 439.627,Z 350.725,A -85,B 0,C 180,E1 -9174.496,E2 -9174.496} C_VEL
LIN {X 0,Y 439.64,Z 350.724,A -85,B 0,C 180,E1 -9178.168,E2 -9178.168} C_VEL
LIN {X 0,Y 439.77,Z 350.708,A -85,B 0,C 180,E1 -9180,E2 -9180} C_VEL
LIN {X 0,Y 439.646,Z 350.722,A -85,B 0,C 180,E1 -9182.749,E2 -9182.749} C_VEL
LIN {X 0,Y 439.624,Z 350.726,A -85,B 0,C 180,E1 -9186.425,E2 -9186.425} C_VEL
LIN {X 0,Y 439.507,Z 350.738,A -85,B 0,C 180,E1 -9189.202,E2 -9189.202} C_VEL
LIN {X 0,Y 439.472,Z 350.741,A -85,B 0,C 180,E1 -9192.938,E2 -9192.938} C_VEL
LIN {X 0,Y 439.454,Z 350.747,A -85,B 0,C 180,E1 -9196.349,E2 -9196.349} C_VEL
LIN {X 0,Y 439.409,Z 350.752,A -85,B 0,C 180,E1 -9199.626,E2 -9199.626} C_VEL
LIN {X 0,Y 439.372,Z 350.754,A -85,B 0,C 180,E1 -9202.575,E2 -9202.575} C_VEL
LIN {X 0,Y 439.412,Z 350.753,A -85,B 0,C 180,E1 -9205.585,E2 -9205.585} C_VEL
LIN {X 0,Y 439.423,Z 350.747,A -85,B 0,C 180,E1 -9208.673,E2 -9208.673} C_VEL
LIN {X 0,Y 439.377,Z 350.756,A -85,B 0,C 180,E1 -9212.03,E2 -9212.03} C_VEL
LIN {X 0,Y 439.401,Z 350.753,A -85,B 0,C 180,E1 -9215.34,E2 -9215.34} C_VEL
LIN {X 0,Y 439.39,Z 350.752,A -85,B 0,C 180,E1 -9218.595,E2 -9218.595} C_VEL
LIN {X 0,Y 439.395,Z 350.754,A -85,B 0,C 180,E1 -9221.257,E2 -9221.257} C_VEL
LIN {X 0,Y 439.408,Z 350.75,A -85,B 0,C 180,E1 -9224.729,E2 -9224.729} C_VEL
LIN {X 0,Y 439.402,Z 350.753,A -85,B 0,C 180,E1 -9227.796,E2 -9227.796} C_VEL
LIN {X 0,Y 439.432,Z 350.747,A -85,B 0,C 180,E1 -9230.227,E2 -9230.227} C_VEL
LIN {X 0,Y 439.378,Z 350.755,A -85,B 0,C 180,E1 -9233.712,E2 -9233.712} C_VEL
LIN {X 0,Y 439.379,Z 350.757,A -85,B 0,C 180,E1 -9237.054,E2 -9237.054} C_VEL
LIN {X 0,Y 439.388,Z 350.752,A -85,B 0,C 180,E1 -9240.274,E2 -9240.274} C_VEL
LIN {X 0,Y 439.435,Z 350.749,A -85,B 0,C 180,E1 -9243.396,E2 -9243.396} C_VEL
LIN {X 0,Y 439.393,Z 350.754,A -85,B 0,C 180,E1 -9246.429,E2 -9246.429} C_VEL
LIN {X 0,Y 439.395,Z 350.753,A -85,B 0,C 180,E1 -9249.397,E2 -9249.397} C_VEL
LIN {X 0,Y 439.437,Z 350.748,A -85,B 0,C 180,E1 -9252.309,E2 -9252.309} C_VEL
LIN {X 0,Y 439.454,Z 350.746,A -85,B 0,C 180,E1 -9255.174,E2 -9255.174} C_VEL
LIN {X 0,Y 439.491,Z 350.74,A -85,B 0,C 180,E1 -9258.001,E2 -9258.001} C_VEL
LIN {X 0,Y 439.54,Z 350.736,A -85,B 0,C 180,E1 -9261.725,E2 -9261.725} C_VEL
LIN {X 0,Y 439.568,Z 350.794,A -85,B 0,C 180,E1 -9262.261,E2 -9262.261} C_VEL
LIN {X 0,Y 442.974,Z 362.726,A -85,B 0,C 180,E1 -9262.937,E2 -9262.937} C_VEL
LIN {X 0,Y 442.597,Z 374.002,A -85,B 0,C 180,E1 -9263.618,E2 -9263.618} C_VEL
LIN {X 0,Y 442.059,Z 385.592,A -85,B 0,C 180,E1 -9264.526,E2 -9264.526} C_VEL
LIN {X 0,Y 441.558,Z 395.947,A -85,B 0,C 180,E1 -9265.549,E2 -9265.549} C_VEL
LIN {X 0,Y 441.266,Z 400.628,A -85,B 0,C 180,E1 -9266.089,E2 -9266.089} C_VEL
LIN {X 0,Y 440.343,Z 404.921,A -85,B 0,C 180,E1 -9266.603,E2 -9266.603} C_VEL
LIN {X 0,Y 437.17,Z 411.611,A -85,B 0,C 180,E1 -9267.465,E2 -9267.465} C_VEL
LIN {X 0,Y 433.984,Z 417.729,A -85,B 0,C 180,E1 -9268.403,E2 -9268.403} C_VEL
LIN {X 0,Y 433.05,Z 421.095,A -85,B 0,C 180,E1 -9269.033,E2 -9269.033} C_VEL
LIN {X 0,Y 432.634,Z 427.319,A -85,B 0,C 180,E1 -9270.465,E2 -9270.465} C_VEL
LIN {X 0,Y 432.416,Z 432.109,A -85,B 0,C 180,E1 -9271.862,E2 -9271.862} C_VEL
LIN {X 0,Y 432.128,Z 435.834,A -85,B 0,C 180,E1 -9273.263,E2 -9273.263} C_VEL
LIN {X 0,Y 432.021,Z 438.547,A -85,B 0,C 180,E1 -9274.665,E2 -9274.665} C_VEL
LIN {X 0,Y 431.924,Z 440.738,A -85,B 0,C 180,E1 -9276.539,E2 -9276.539} C_VEL
LIN {X 0,Y 431.94,Z 441.24,A -85,B 0,C 180,E1 -9277.479,E2 -9277.479} C_VEL
LIN {X 0,Y 431.924,Z 441.047,A -85,B 0,C 180,E1 -9279.364,E2 -9279.364} C_VEL
LIN {X 0,Y 431.949,Z 440.382,A -85,B 0,C 180,E1 -9280.309,E2 -9280.309} C_VEL
LIN {X 0,Y 432.016,Z 439.297,A -85,B 0,C 180,E1 -9281.257,E2 -9281.257} C_VEL
LIN {X 0,Y 432.291,Z 436.786,A -85,B 0,C 180,E1 -9282.718,E2 -9282.718} C_VEL
LIN {X 0,Y 432.528,Z 433.444,A -85,B 0,C 180,E1 -9284.106,E2 -9284.106} C_VEL
LIN {X 0,Y 432.857,Z 428.885,A -85,B 0,C 180,E1 -9285.539,E2 -9285.539} C_VEL
LIN {X 0,Y 433.382,Z 421.932,A -85,B 0,C 180,E1 -9287.214,E2 -9287.214} C_VEL
LIN {X 0,Y 433.949,Z 414.335,A -85,B 0,C 180,E1 -9288.654,E2 -9288.654} C_VEL
LIN {X 0,Y 434.66,Z 405.202,A -85,B 0,C 180,E1 -9290.023,E2 -9290.023} C_VEL
LIN {X 0,Y 435.237,Z 395.714,A -85,B 0,C 180,E1 -9291.179,E2 -9291.179} C_VEL
LIN {X 0,Y 435.788,Z 385.952,A -85,B 0,C 180,E1 -9292.145,E2 -9292.145} C_VEL
LIN {X 0,Y 436.449,Z 374.826,A -85,B 0,C 180,E1 -9293.018,E2 -9293.018} C_VEL
LIN {X 0,Y 436.85,Z 366.27,A -85,B 0,C 180,E1 -9293.558,E2 -9293.558} C_VEL
LIN {X 0,Y 434.35,Z 357.64,A -85,B 0,C 180,E1 -9294.136,E2 -9294.136} C_VEL
LIN {X 0,Y 432.382,Z 351.628,A -85,B 0,C 180,E1 -9294.522,E2 -9294.522} C_VEL
LIN {X 0,Y 432.393,Z 351.627,A -85,B 0,C 180,E1 -9297.071,E2 -9297.071} C_VEL
LIN {X 0,Y 432.349,Z 351.633,A -85,B 0,C 180,E1 -9300.51,E2 -9300.51} C_VEL
LIN {X 0,Y 432.36,Z 351.629,A -85,B 0,C 180,E1 -9304.003,E2 -9304.003} C_VEL
LIN {X 0,Y 432.323,Z 351.637,A -85,B 0,C 180,E1 -9307.196,E2 -9307.196} C_VEL
LIN {X 0,Y 432.337,Z 351.632,A -85,B 0,C 180,E1 -9310.179,E2 -9310.179} C_VEL
LIN {X 0,Y 432.323,Z 351.635,A -85,B 0,C 180,E1 -9313.059,E2 -9313.059} C_VEL
LIN {X 0,Y 432.332,Z 351.635,A -85,B 0,C 180,E1 -9315.664,E2 -9315.664} C_VEL
LIN {X 0,Y 432.366,Z 351.632,A -85,B 0,C 180,E1 -9318.392,E2 -9318.392} C_VEL
LIN {X 0,Y 432.353,Z 351.632,A -85,B 0,C 180,E1 -9321.851,E2 -9321.851} C_VEL
LIN {X 0,Y 432.34,Z 351.634,A -85,B 0,C 180,E1 -9325.322,E2 -9325.322} C_VEL
LIN {X 0,Y 432.328,Z 351.621,A -85,B 0,C 180,E1 -9328.654,E2 -9328.654} C_VEL
LIN {X 0,Y 432.379,Z 351.615,A -85,B 0,C 180,E1 -9331.368,E2 -9331.368} C_VEL
LIN {X 0,Y 432.362,Z 351.628,A -85,B 0,C 180,E1 -9333.967,E2 -9333.967} C_VEL
LIN {X 0,Y 432.317,Z 351.628,A -85,B 0,C 180,E1 -9337.035,E2 -9337.035} C_VEL
LIN {X 0,Y 432.384,Z 351.626,A -85,B 0,C 180,E1 -9340.514,E2 -9340.514} C_VEL
LIN {X 0,Y 432.428,Z 351.62,A -85,B 0,C 180,E1 -9343.961,E2 -9343.961} C_VEL
LIN {X 0,Y 432.479,Z 351.615,A -85,B 0,C 180,E1 -9347.804,E2 -9347.804} C_VEL
LIN {X 0,Y 432.489,Z 351.614,A -85,B 0,C 180,E1 -9351.59,E2 -9351.59} C_VEL
LIN {X 0,Y 432.595,Z 351.594,A -85,B 0,C 180,E1 -9354.406,E2 -9354.406} C_VEL
LIN {X 0,Y 432.603,Z 351.6,A -85,B 0,C 180,E1 -9358.138,E2 -9358.138} C_VEL
LIN {X 0,Y 432.732,Z 351.577,A -85,B 0,C 180,E1 -9360,E2 -9360} C_VEL
LIN {X 0,Y 432.603,Z 351.6,A -85,B 0,C 180,E1 -9362.793,E2 -9362.793} C_VEL
LIN {X 0,Y 432.569,Z 351.604,A -85,B 0,C 180,E1 -9366.53,E2 -9366.53} C_VEL
LIN {X 0,Y 432.439,Z 351.616,A -85,B 0,C 180,E1 -9369.353,E2 -9369.353} C_VEL
LIN {X 0,Y 432.426,Z 351.62,A -85,B 0,C 180,E1 -9372.804,E2 -9372.804} C_VEL
LIN {X 0,Y 432.409,Z 351.623,A -85,B 0,C 180,E1 -9376.479,E2 -9376.479} C_VEL
LIN {X 0,Y 432.335,Z 351.634,A -85,B 0,C 180,E1 -9379.961,E2 -9379.961} C_VEL
LIN {X 0,Y 432.316,Z 351.637,A -85,B 0,C 180,E1 -9382.964,E2 -9382.964} C_VEL
LIN {X 0,Y 432.361,Z 351.632,A -85,B 0,C 180,E1 -9386.033,E2 -9386.033} C_VEL
LIN {X 0,Y 432.349,Z 351.635,A -85,B 0,C 180,E1 -9389.187,E2 -9389.187} C_VEL
LIN {X 0,Y 432.322,Z 351.637,A -85,B 0,C 180,E1 -9392.294,E2 -9392.294} C_VEL
LIN {X 0,Y 432.338,Z 351.633,A -85,B 0,C 180,E1 -9394.677,E2 -9394.677} C_VEL
LIN {X 0,Y 432.351,Z 351.625,A -85,B 0,C 180,E1 -9398.149,E2 -9398.149} C_VEL
LIN {X 0,Y 432.37,Z 351.622,A -85,B 0,C 180,E1 -9401.609,E2 -9401.609} C_VEL
LIN {X 0,Y 432.375,Z 351.623,A -85,B 0,C 180,E1 -9404.342,E2 -9404.342} C_VEL
LIN {X 0,Y 432.393,Z 351.8,A -85,B 0,C 180,E1 -9407.72,E2 -9407.72} C_VEL
LIN {X 0,Y 433.789,Z 358.665,A -85,B 0,C 180,E1 -9410.249,E2 -9410.249} C_VEL
LIN {X 0,Y 435.157,Z 366.145,A -85,B 0,C 180,E1 -9412.845,E2 -9412.845} C_VEL
LIN {X 0,Y 435.309,Z 369.167,A -85,B 0,C 180,E1 -9413.828,E2 -9413.828} C_VEL
LIN {X 0,Y 434.331,Z 380.513,A -85,B 0,C 180,E1 -9417.291,E2 -9417.291} C_VEL
LIN {X 0,Y 433.687,Z 391.003,A -85,B 0,C 180,E1 -9420.38,E2 -9420.38} C_VEL
LIN {X 0,Y 433.073,Z 402.258,A -85,B 0,C 180,E1 -9423.597,E2 -9423.597} C_VEL
LIN {X 0,Y 432.511,Z 414.624,A -85,B 0,C 180,E1 -9427.047,E2 -9427.047} C_VEL
LIN {X 0,Y 432.078,Z 426.815,A -85,B 0,C 180,E1 -9430.391,E2 -9430.391} C_VEL
LIN {X 0,Y 431.825,Z 436.686,A -85,B 0,C 180,E1 -9433.07,E2 -9433.07} C_VEL
LIN {X 0,Y 433.859,Z 452.623,A -85,B 0,C 180,E1 -9433.611,E2 -9433.611} C_VEL
LIN {X 0,Y 434.719,Z 465.734,A -85,B 0,C 180,E1 -9434.229,E2 -9434.229} C_VEL
LIN {X 0,Y 435.047,Z 471.124,A -85,B 0,C 180,E1 -9434.542,E2 -9434.542} C_VEL
LIN {X 0,Y 434.269,Z 483.405,A -85,B 0,C 180,E1 -9435.353,E2 -9435.353} C_VEL
LIN {X 0,Y 433.545,Z 494.778,A -85,B 0,C 180,E1 -9436.322,E2 -9436.322} C_VEL
LIN {X 0,Y 433.069,Z 504.425,A -85,B 0,C 180,E1 -9437.346,E2 -9437.346} C_VEL
LIN {X 0,Y 432.427,Z 513.541,A -85,B 0,C 180,E1 -9438.517,E2 -9438.517} C_VEL
LIN {X 0,Y 431.888,Z 522.484,A -85,B 0,C 180,E1 -9439.926,E2 -9439.926} C_VEL
LIN {X 0,Y 431.695,Z 529.695,A -85,B 0,C 180,E1 -9441.34,E2 -9441.34} C_VEL
LIN {X 0,Y 431.527,Z 536.314,A -85,B 0,C 180,E1 -9442.985,E2 -9442.985} C_VEL
LIN {X 0,Y 431.551,Z 540.709,A -85,B 0,C 180,E1 -9444.393,E2 -9444.393} C_VEL
LIN {X 0,Y 431.55,Z 543.045,A -85,B 0,C 180,E1 -9445.33,E2 -9445.33} C_VEL
LIN {X 0,Y 431.648,Z 544.926,A -85,B 0,C 180,E1 -9446.267,E2 -9446.267} C_VEL
LIN {X 0,Y 431.617,Z 546.336,A -85,B 0,C 180,E1 -9447.201,E2 -9447.201} C_VEL
LIN {X 0,Y 431.583,Z 547.952,A -85,B 0,C 180,E1 -9449.068,E2 -9449.068} C_VEL
LIN {X 0,Y 431.607,Z 548.141,A -85,B 0,C 180,E1 -9450.001,E2 -9450.001} C_VEL
LIN {X 0,Y 431.59,Z 547.896,A -85,B 0,C 180,E1 -9450.934,E2 -9450.934} C_VEL
LIN {X 0,Y 431.592,Z 547.256,A -85,B 0,C 180,E1 -9451.867,E2 -9451.867} C_VEL
LIN {X 0,Y 431.621,Z 546.219,A -85,B 0,C 180,E1 -9452.801,E2 -9452.801} C_VEL
LIN {X 0,Y 431.706,Z 544.749,A -85,B 0,C 180,E1 -9453.734,E2 -9453.734} C_VEL
LIN {X 0,Y 431.531,Z 541.665,A -85,B 0,C 180,E1 -9455.14,E2 -9455.14} C_VEL
LIN {X 0,Y 431.564,Z 537.356,A -85,B 0,C 180,E1 -9456.594,E2 -9456.594} C_VEL
LIN {X 0,Y 431.672,Z 531.149,A -85,B 0,C 180,E1 -9458.191,E2 -9458.191} C_VEL
LIN {X 0,Y 431.819,Z 524.209,A -85,B 0,C 180,E1 -9459.604,E2 -9459.604} C_VEL
LIN {X 0,Y 432.237,Z 515.611,A -85,B 0,C 180,E1 -9461.015,E2 -9461.015} C_VEL
LIN {X 0,Y 432.699,Z 506.761,A -85,B 0,C 180,E1 -9462.19,E2 -9462.19} C_VEL
LIN {X 0,Y 433.237,Z 496.118,A -85,B 0,C 180,E1 -9463.342,E2 -9463.342} C_VEL
LIN {X 0,Y 433.934,Z 485.09,A -85,B 0,C 180,E1 -9464.3,E2 -9464.3} C_VEL
LIN {X 0,Y 434.591,Z 473.023,A -85,B 0,C 180,E1 -9465.116,E2 -9465.116} C_VEL
LIN {X 0,Y 434.591,Z 467.742,A -85,B 0,C 180,E1 -9465.416,E2 -9465.416} C_VEL
LIN {X 0,Y 433.498,Z 454.129,A -85,B 0,C 180,E1 -9466.061,E2 -9466.061} C_VEL
LIN {X 0,Y 432.18,Z 441.221,A -85,B 0,C 180,E1 -9466.488,E2 -9466.488} C_VEL
LIN {X 0,Y 431.776,Z 437.244,A -85,B 0,C 180,E1 -9466.59,E2 -9466.59} C_VEL
LIN {X 0,Y 432.11,Z 424.595,A -85,B 0,C 180,E1 -9469.972,E2 -9469.972} C_VEL
LIN {X 0,Y 432.429,Z 413.508,A -85,B 0,C 180,E1 -9472.959,E2 -9472.959} C_VEL
LIN {X 0,Y 432.837,Z 402.31,A -85,B 0,C 180,E1 -9476.003,E2 -9476.003} C_VEL
LIN {X 0,Y 433.391,Z 391.074,A -85,B 0,C 180,E1 -9479.111,E2 -9479.111} C_VEL
LIN {X 0,Y 434.02,Z 378.61,A -85,B 0,C 180,E1 -9482.645,E2 -9482.645} C_VEL
LIN {X 0,Y 434.826,Z 366.85,A -85,B 0,C 180,E1 -9486.085,E2 -9486.085} C_VEL
LIN {X 0,Y 434.338,Z 362.18,A -85,B 0,C 180,E1 -9487.546,E2 -9487.546} C_VEL
LIN {X 0,Y 432.663,Z 353.145,A -85,B 0,C 180,E1 -9490.523,E2 -9490.523} C_VEL
LIN {X 0,Y 432.355,Z 351.632,A -85,B 0,C 180,E1 -9491.097,E2 -9491.097} C_VEL
LIN {X 0,Y 432.345,Z 351.634,A -85,B 0,C 180,E1 -9494.347,E2 -9494.347} C_VEL
LIN {X 0,Y 432.324,Z 351.635,A -85,B 0,C 180,E1 -9497.016,E2 -9497.016} C_VEL
LIN {X 0,Y 432.341,Z 351.629,A -85,B 0,C 180,E1 -9499.821,E2 -9499.821} C_VEL
LIN {X 0,Y 432.311,Z 351.637,A -85,B 0,C 180,E1 -9503.022,E2 -9503.022} C_VEL
LIN {X 0,Y 432.364,Z 351.627,A -85,B 0,C 180,E1 -9505.997,E2 -9505.997} C_VEL
LIN {X 0,Y 432.353,Z 351.629,A -85,B 0,C 180,E1 -9509.49,E2 -9509.49} C_VEL
LIN {X 0,Y 432.396,Z 351.627,A -85,B 0,C 180,E1 -9512.929,E2 -9512.929} C_VEL
LIN {X 0,Y 432.377,Z 351.626,A -85,B 0,C 180,E1 -9516.024,E2 -9516.024} C_VEL
LIN {X 0,Y 432.355,Z 351.63,A -85,B 0,C 180,E1 -9519.046,E2 -9519.046} C_VEL
LIN {X 0,Y 432.379,Z 351.626,A -85,B 0,C 180,E1 -9522.011,E2 -9522.011} C_VEL
LIN {X 0,Y 432.401,Z 351.625,A -85,B 0,C 180,E1 -9524.927,E2 -9524.927} C_VEL
LIN {X 0,Y 432.465,Z 351.616,A -85,B 0,C 180,E1 -9527.804,E2 -9527.804} C_VEL
LIN {X 0,Y 432.497,Z 351.61,A -85,B 0,C 180,E1 -9531.591,E2 -9531.591} C_VEL
LIN {X 0,Y 432.603,Z 351.601,A -85,B 0,C 180,E1 -9534.406,E2 -9534.406} C_VEL
LIN {X 0,Y 432.61,Z 351.6,A -85,B 0,C 180,E1 -9538.138,E2 -9538.138} C_VEL
LIN {X 0,Y 432.74,Z 351.584,A -85,B 0,C 180,E1 -9540,E2 -9540} C_VEL
LIN {X 0,Y 432.598,Z 351.599,A -85,B 0,C 180,E1 -9542.794,E2 -9542.794} C_VEL
LIN {X 0,Y 432.579,Z 351.602,A -85,B 0,C 180,E1 -9546.53,E2 -9546.53} C_VEL
LIN {X 0,Y 432.449,Z 351.617,A -85,B 0,C 180,E1 -9549.353,E2 -9549.353} C_VEL
LIN {X 0,Y 432.437,Z 351.618,A -85,B 0,C 180,E1 -9552.804,E2 -9552.804} C_VEL
LIN {X 0,Y 432.419,Z 351.622,A -85,B 0,C 180,E1 -9556.479,E2 -9556.479} C_VEL
LIN {X 0,Y 432.345,Z 351.634,A -85,B 0,C 180,E1 -9559.96,E2 -9559.96} C_VEL
LIN {X 0,Y 432.326,Z 351.631,A -85,B 0,C 180,E1 -9562.964,E2 -9562.964} C_VEL
LIN {X 0,Y 432.371,Z 351.629,A -85,B 0,C 180,E1 -9566.032,E2 -9566.032} C_VEL
LIN {X 0,Y 432.349,Z 351.631,A -85,B 0,C 180,E1 -9569.187,E2 -9569.187} C_VEL
LIN {X 0,Y 432.329,Z 351.632,A -85,B 0,C 180,E1 -9572.443,E2 -9572.443} C_VEL
LIN {X 0,Y 432.35,Z 351.633,A -85,B 0,C 180,E1 -9575.632,E2 -9575.632} C_VEL
LIN {X 0,Y 432.357,Z 351.632,A -85,B 0,C 180,E1 -9579.343,E2 -9579.343} C_VEL
LIN {X 0,Y 432.34,Z 351.632,A -85,B 0,C 180,E1 -9581.797,E2 -9581.797} C_VEL
LIN {X 0,Y 432.34,Z 351.63,A -85,B 0,C 180,E1 -9584.347,E2 -9584.347} C_VEL
LIN {X 0,Y 432.327,Z 351.634,A -85,B 0,C 180,E1 -9587.015,E2 -9587.015} C_VEL
LIN {X 0,Y 432.34,Z 351.632,A -85,B 0,C 180,E1 -9589.821,E2 -9589.821} C_VEL
LIN {X 0,Y 432.311,Z 351.637,A -85,B 0,C 180,E1 -9593.022,E2 -9593.022} C_VEL
LIN {X 0,Y 432.366,Z 351.627,A -85,B 0,C 180,E1 -9595.996,E2 -9595.996} C_VEL
LIN {X 0,Y 432.354,Z 351.63,A -85,B 0,C 180,E1 -9599.489,E2 -9599.489} C_VEL
LIN {X 0,Y 432.398,Z 351.627,A -85,B 0,C 180,E1 -9602.928,E2 -9602.928} C_VEL
LIN {X 0,Y 432.378,Z 351.625,A -85,B 0,C 180,E1 -9606.023,E2 -9606.023} C_VEL
LIN {X 0,Y 432.357,Z 351.631,A -85,B 0,C 180,E1 -9609.046,E2 -9609.046} C_VEL
LIN {X 0,Y 432.384,Z 351.625,A -85,B 0,C 180,E1 -9612.011,E2 -9612.011} C_VEL
LIN {X 0,Y 432.402,Z 351.626,A -85,B 0,C 180,E1 -9614.926,E2 -9614.926} C_VEL
LIN {X 0,Y 432.466,Z 351.614,A -85,B 0,C 180,E1 -9617.803,E2 -9617.803} C_VEL
LIN {X 0,Y 432.524,Z 351.611,A -85,B 0,C 180,E1 -9621.813,E2 -9621.813} C_VEL
LIN {X 0,Y 432.558,Z 351.786,A -85,B 0,C 180,E1 -9622.036,E2 -9622.036} C_VEL
LIN {X 0,Y 436.102,Z 364.394,A -85,B 0,C 180,E1 -9622.766,E2 -9622.766} C_VEL
LIN {X 0,Y 435.665,Z 376.253,A -85,B 0,C 180,E1 -9623.516,E2 -9623.516} C_VEL
LIN {X 0,Y 435.096,Z 387.556,A -85,B 0,C 180,E1 -9624.438,E2 -9624.438} C_VEL
LIN {X 0,Y 434.564,Z 397.728,A -85,B 0,C 180,E1 -9625.477,E2 -9625.477} C_VEL
LIN {X 0,Y 434.06,Z 406.059,A -85,B 0,C 180,E1 -9626.518,E2 -9626.518} C_VEL
LIN {X 0,Y 433.567,Z 413.749,A -85,B 0,C 180,E1 -9627.677,E2 -9627.677} C_VEL
LIN {X 0,Y 433.05,Z 421.095,A -85,B 0,C 180,E1 -9629.033,E2 -9629.033} C_VEL
LIN {X 0,Y 432.136,Z 424.259,A -85,B 0,C 180,E1 -9629.683,E2 -9629.683} C_VEL
LIN {X 0,Y 429.041,Z 429.062,A -85,B 0,C 180,E1 -9630.762,E2 -9630.762} C_VEL
LIN {X 0,Y 426.005,Z 433.216,A -85,B 0,C 180,E1 -9631.899,E2 -9631.899} C_VEL
LIN {X 0,Y 425.196,Z 435.313,A -85,B 0,C 180,E1 -9632.634,E2 -9632.634} C_VEL
LIN {X 0,Y 424.991,Z 437.938,A -85,B 0,C 180,E1 -9633.792,E2 -9633.792} C_VEL
LIN {X 0,Y 424.993,Z 439.569,A -85,B 0,C 180,E1 -9634.742,E2 -9634.742} C_VEL
LIN {X 0,Y 424.888,Z 441.692,A -85,B 0,C 180,E1 -9636.648,E2 -9636.648} C_VEL
LIN {X 0,Y 424.908,Z 442.13,A -85,B 0,C 180,E1 -9637.603,E2 -9637.603} C_VEL
LIN {X 0,Y 424.894,Z 441.872,A -85,B 0,C 180,E1 -9639.52,E2 -9639.52} C_VEL
LIN {X 0,Y 424.933,Z 441.168,A -85,B 0,C 180,E1 -9640.481,E2 -9640.481} C_VEL
LIN {X 0,Y 425.02,Z 440.018,A -85,B 0,C 180,E1 -9641.444,E2 -9641.444} C_VEL
LIN {X 0,Y 425.281,Z 437.648,A -85,B 0,C 180,E1 -9642.834,E2 -9642.834} C_VEL
LIN {X 0,Y 425.567,Z 434.021,A -85,B 0,C 180,E1 -9644.342,E2 -9644.342} C_VEL
LIN {X 0,Y 425.937,Z 429.378,A -85,B 0,C 180,E1 -9645.798,E2 -9645.798} C_VEL
LIN {X 0,Y 426.437,Z 423.446,A -85,B 0,C 180,E1 -9647.256,E2 -9647.256} C_VEL
LIN {X 0,Y 427.025,Z 416.001,A -85,B 0,C 180,E1 -9648.719,E2 -9648.719} C_VEL
LIN {X 0,Y 427.664,Z 408.338,A -85,B 0,C 180,E1 -9649.937,E2 -9649.937} C_VEL
LIN {X 0,Y 428.3,Z 398.917,A -85,B 0,C 180,E1 -9651.161,E2 -9651.161} C_VEL
LIN {X 0,Y 428.976,Z 388.346,A -85,B 0,C 180,E1 -9652.262,E2 -9652.262} C_VEL
LIN {X 0,Y 429.698,Z 376.695,A -85,B 0,C 180,E1 -9653.222,E2 -9653.222} C_VEL
LIN {X 0,Y 430.087,Z 367.341,A -85,B 0,C 180,E1 -9653.832,E2 -9653.832} C_VEL
LIN {X 0,Y 426.596,Z 356.376,A -85,B 0,C 180,E1 -9654.588,E2 -9654.588} C_VEL
LIN {X 0,Y 425.333,Z 352.506,A -85,B 0,C 180,E1 -9654.836,E2 -9654.836} C_VEL
LIN {X 0,Y 425.351,Z 352.506,A -85,B 0,C 180,E1 -9657.557,E2 -9657.557} C_VEL
LIN {X 0,Y 425.289,Z 352.511,A -85,B 0,C 180,E1 -9660.815,E2 -9660.815} C_VEL
LIN {X 0,Y 425.312,Z 352.507,A -85,B 0,C 180,E1 -9664.287,E2 -9664.287} C_VEL
LIN {X 0,Y 425.28,Z 352.512,A -85,B 0,C 180,E1 -9667.693,E2 -9667.693} C_VEL
LIN {X 0,Y 425.282,Z 352.513,A -85,B 0,C 180,E1 -9670.52,E2 -9670.52} C_VEL
LIN {X 0,Y 425.263,Z 352.515,A -85,B 0,C 180,E1 -9673.351,E2 -9673.351} C_VEL
LIN {X 0,Y 425.257,Z 352.514,A -85,B 0,C 180,E1 -9676.648,E2 -9676.648} C_VEL
LIN {X 0,Y 425.299,Z 352.51,A -85,B 0,C 180,E1 -9679.476,E2 -9679.476} C_VEL
LIN {X 0,Y 425.286,Z 352.513,A -85,B 0,C 180,E1 -9682.486,E2 -9682.486} C_VEL
LIN {X 0,Y 425.306,Z 352.509,A -85,B 0,C 180,E1 -9685.817,E2 -9685.817} C_VEL
LIN {X 0,Y 425.3,Z 352.49,A -85,B 0,C 180,E1 -9689.235,E2 -9689.235} C_VEL
LIN {X 0,Y 425.348,Z 352.497,A -85,B 0,C 180,E1 -9692.442,E2 -9692.442} C_VEL
LIN {X 0,Y 425.349,Z 352.501,A -85,B 0,C 180,E1 -9695.602,E2 -9695.602} C_VEL
LIN {X 0,Y 425.291,Z 352.51,A -85,B 0,C 180,E1 -9698.681,E2 -9698.681} C_VEL
LIN {X 0,Y 425.331,Z 352.5,A -85,B 0,C 180,E1 -9701.702,E2 -9701.702} C_VEL
LIN {X 0,Y 425.346,Z 352.504,A -85,B 0,C 180,E1 -9704.67,E2 -9704.67} C_VEL
LIN {X 0,Y 425.428,Z 352.494,A -85,B 0,C 180,E1 -9707.598,E2 -9707.598} C_VEL
LIN {X 0,Y 425.44,Z 352.493,A -85,B 0,C 180,E1 -9711.45,E2 -9711.45} C_VEL
LIN {X 0,Y 425.552,Z 352.471,A -85,B 0,C 180,E1 -9714.313,E2 -9714.313} C_VEL
LIN {X 0,Y 425.573,Z 352.476,A -85,B 0,C 180,E1 -9718.107,E2 -9718.107} C_VEL
LIN {X 0,Y 425.702,Z 352.452,A -85,B 0,C 180,E1 -9720,E2 -9720} C_VEL
LIN {X 0,Y 425.554,Z 352.478,A -85,B 0,C 180,E1 -9722.84,E2 -9722.84} C_VEL
LIN {X 0,Y 425.528,Z 352.48,A -85,B 0,C 180,E1 -9726.639,E2 -9726.639} C_VEL
LIN {X 0,Y 425.398,Z 352.492,A -85,B 0,C 180,E1 -9729.509,E2 -9729.509} C_VEL
LIN {X 0,Y 425.389,Z 352.497,A -85,B 0,C 180,E1 -9732.904,E2 -9732.904} C_VEL
LIN {X 0,Y 425.357,Z 352.501,A -85,B 0,C 180,E1 -9736.605,E2 -9736.605} C_VEL
LIN {X 0,Y 425.325,Z 352.506,A -85,B 0,C 180,E1 -9739.636,E2 -9739.636} C_VEL
LIN {X 0,Y 425.303,Z 352.508,A -85,B 0,C 180,E1 -9743.365,E2 -9743.365} C_VEL
LIN {X 0,Y 425.345,Z 352.506,A -85,B 0,C 180,E1 -9746.845,E2 -9746.845} C_VEL
LIN {X 0,Y 425.315,Z 352.509,A -85,B 0,C 180,E1 -9749.718,E2 -9749.718} C_VEL
LIN {X 0,Y 425.279,Z 352.514,A -85,B 0,C 180,E1 -9753.048,E2 -9753.048} C_VEL
LIN {X 0,Y 425.282,Z 352.51,A -85,B 0,C 180,E1 -9755.93,E2 -9755.93} C_VEL
LIN {X 0,Y 425.311,Z 352.502,A -85,B 0,C 180,E1 -9759.047,E2 -9759.047} C_VEL
LIN {X 0,Y 425.329,Z 352.507,A -85,B 0,C 180,E1 -9762.646,E2 -9762.646} C_VEL
LIN {X 0,Y 425.316,Z 352.504,A -85,B 0,C 180,E1 -9766.052,E2 -9766.052} C_VEL
LIN {X 0,Y 425.323,Z 352.527,A -85,B 0,C 180,E1 -9767.283,E2 -9767.283} C_VEL
LIN {X 0,Y 426.811,Z 359.853,A -85,B 0,C 180,E1 -9770.046,E2 -9770.046} C_VEL
LIN {X 0,Y 428.144,Z 367.06,A -85,B 0,C 180,E1 -9772.602,E2 -9772.602} C_VEL
LIN {X 0,Y 428.358,Z 370.662,A -85,B 0,C 180,E1 -9773.798,E2 -9773.798} C_VEL
LIN {X 0,Y 427.252,Z 383.198,A -85,B 0,C 180,E1 -9777.684,E2 -9777.684} C_VEL
LIN {X 0,Y 426.47,Z 394.804,A -85,B 0,C 180,E1 -9781.144,E2 -9781.144} C_VEL
LIN {X 0,Y 425.927,Z 404.89,A -85,B 0,C 180,E1 -9784.071,E2 -9784.071} C_VEL
LIN {X 0,Y 425.378,Z 417.554,A -85,B 0,C 180,E1 -9787.667,E2 -9787.667} C_VEL
LIN {X 0,Y 424.932,Z 430.162,A -85,B 0,C 180,E1 -9791.186,E2 -9791.186} C_VEL
LIN {X 0,Y 424.757,Z 435.826,A -85,B 0,C 180,E1 -9792.757,E2 -9792.757} C_VEL
LIN {X 0,Y 426.788,Z 450.656,A -85,B 0,C 180,E1 -9793.259,E2 -9793.259} C_VEL
LIN {X 0,Y 427.656,Z 463.181,A -85,B 0,C 180,E1 -9793.839,E2 -9793.839} C_VEL
LIN {X 0,Y 428.097,Z 472.759,A -85,B 0,C 180,E1 -9794.406,E2 -9794.406} C_VEL
LIN {X 0,Y 427.273,Z 484.422,A -85,B 0,C 180,E1 -9795.23,E2 -9795.23} C_VEL
LIN {X 0,Y 426.503,Z 495.494,A -85,B 0,C 180,E1 -9796.226,E2 -9796.226} C_VEL
LIN {X 0,Y 425.935,Z 505.778,A -85,B 0,C 180,E1 -9797.375,E2 -9797.375} C_VEL
LIN {X 0,Y 425.315,Z 514.503,A -85,B 0,C 180,E1 -9798.564,E2 -9798.564} C_VEL
LIN {X 0,Y 424.792,Z 523.038,A -85,B 0,C 180,E1 -9799.997,E2 -9799.997} C_VEL
LIN {X 0,Y 424.618,Z 529.963,A -85,B 0,C 180,E1 -9801.434,E2 -9801.434} C_VEL
LIN {X 0,Y 424.441,Z 535.518,A -85,B 0,C 180,E1 -9802.867,E2 -9802.867} C_VEL
LIN {X 0,Y 424.486,Z 539.897,A -85,B 0,C 180,E1 -9804.3,E2 -9804.3} C_VEL
LIN {X 0,Y 424.464,Z 542.222,A -85,B 0,C 180,E1 -9805.252,E2 -9805.252} C_VEL
LIN {X 0,Y 424.576,Z 544.086,A -85,B 0,C 180,E1 -9806.204,E2 -9806.204} C_VEL
LIN {X 0,Y 424.568,Z 545.491,A -85,B 0,C 180,E1 -9807.154,E2 -9807.154} C_VEL
LIN {X 0,Y 424.533,Z 547.091,A -85,B 0,C 180,E1 -9809.052,E2 -9809.052} C_VEL
LIN {X 0,Y 424.562,Z 547.264,A -85,B 0,C 180,E1 -9810.001,E2 -9810.001} C_VEL
LIN {X 0,Y 424.543,Z 547.01,A -85,B 0,C 180,E1 -9810.949,E2 -9810.949} C_VEL
LIN {X 0,Y 424.543,Z 546.362,A -85,B 0,C 180,E1 -9811.898,E2 -9811.898} C_VEL
LIN {X 0,Y 424.574,Z 545.316,A -85,B 0,C 180,E1 -9812.847,E2 -9812.847} C_VEL
LIN {X 0,Y 424.645,Z 543.826,A -85,B 0,C 180,E1 -9813.797,E2 -9813.797} C_VEL
LIN {X 0,Y 424.466,Z 540.721,A -85,B 0,C 180,E1 -9815.226,E2 -9815.226} C_VEL
LIN {X 0,Y 424.5,Z 536.555,A -85,B 0,C 180,E1 -9816.656,E2 -9816.656} C_VEL
LIN {X 0,Y 424.601,Z 530.151,A -85,B 0,C 180,E1 -9818.328,E2 -9818.328} C_VEL
LIN {X 0,Y 424.764,Z 523.18,A -85,B 0,C 180,E1 -9819.765,E2 -9819.765} C_VEL
LIN {X 0,Y 425.197,Z 514.53,A -85,B 0,C 180,E1 -9821.199,E2 -9821.199} C_VEL
LIN {X 0,Y 425.738,Z 505.643,A -85,B 0,C 180,E1 -9822.393,E2 -9822.393} C_VEL
LIN {X 0,Y 426.289,Z 494.7,A -85,B 0,C 180,E1 -9823.588,E2 -9823.588} C_VEL
LIN {X 0,Y 426.95,Z 483.817,A -85,B 0,C 180,E1 -9824.539,E2 -9824.539} C_VEL
LIN {X 0,Y 427.673,Z 471.625,A -85,B 0,C 180,E1 -9825.367,E2 -9825.367} C_VEL
LIN {X 0,Y 426.976,Z 459.931,A -85,B 0,C 180,E1 -9826.005,E2 -9826.005} C_VEL
LIN {X 0,Y 425.822,Z 447.079,A -85,B 0,C 180,E1 -9826.531,E2 -9826.531} C_VEL
LIN {X 0,Y 424.732,Z 436.42,A -85,B 0,C 180,E1 -9826.835,E2 -9826.835} C_VEL
LIN {X 0,Y 425.045,Z 423.641,A -85,B 0,C 180,E1 -9830.319,E2 -9830.319} C_VEL
LIN {X 0,Y 425.423,Z 412.588,A -85,B 0,C 180,E1 -9833.359,E2 -9833.359} C_VEL
LIN {X 0,Y 425.969,Z 399.468,A -85,B 0,C 180,E1 -9837.009,E2 -9837.009} C_VEL
LIN {X 0,Y 426.514,Z 388.327,A -85,B 0,C 180,E1 -9840.171,E2 -9840.171} C_VEL
LIN {X 0,Y 427.15,Z 377.073,A -85,B 0,C 180,E1 -9843.448,E2 -9843.448} C_VEL
LIN {X 0,Y 427.851,Z 367.214,A -85,B 0,C 180,E1 -9846.4,E2 -9846.4} C_VEL
LIN {X 0,Y 427.003,Z 361.496,A -85,B 0,C 180,E1 -9848.241,E2 -9848.241} C_VEL
LIN {X 0,Y 425.333,Z 352.505,A -85,B 0,C 180,E1 -9851.319,E2 -9851.319} C_VEL
LIN {X 0,Y 425.294,Z 352.513,A -85,B 0,C 180,E1 -9854.718,E2 -9854.718} C_VEL
LIN {X 0,Y 425.294,Z 352.507,A -85,B 0,C 180,E1 -9858.042,E2 -9858.042} C_VEL
LIN {X 0,Y 425.314,Z 352.508,A -85,B 0,C 180,E1 -9861.103,E2 -9861.103} C_VEL
LIN {X 0,Y 425.304,Z 352.509,A -85,B 0,C 180,E1 -9864.665,E2 -9864.665} C_VEL
LIN {X 0,Y 425.27,Z 352.51,A -85,B 0,C 180,E1 -9868.074,E2 -9868.074} C_VEL
LIN {X 0,Y 425.336,Z 352.504,A -85,B 0,C 180,E1 -9871.368,E2 -9871.368} C_VEL
LIN {X 0,Y 425.301,Z 352.51,A -85,B 0,C 180,E1 -9874.555,E2 -9874.555} C_VEL
LIN {X 0,Y 425.293,Z 352.508,A -85,B 0,C 180,E1 -9877.662,E2 -9877.662} C_VEL
LIN {X 0,Y 425.366,Z 352.503,A -85,B 0,C 180,E1 -9880.704,E2 -9880.704} C_VEL
LIN {X 0,Y 425.393,Z 352.495,A -85,B 0,C 180,E1 -9883.689,E2 -9883.689} C_VEL
LIN {X 0,Y 425.417,Z 352.492,A -85,B 0,C 180,E1 -9887.599,E2 -9887.599} C_VEL
LIN {X 0,Y 425.448,Z 352.488,A -85,B 0,C 180,E1 -9891.45,E2 -9891.45} C_VEL
LIN {X 0,Y 425.56,Z 352.479,A -85,B 0,C 180,E1 -9894.314,E2 -9894.314} C_VEL
LIN {X 0,Y 425.579,Z 352.476,A -85,B 0,C 180,E1 -9898.107,E2 -9898.107} C_VEL
LIN {X 0,Y 425.71,Z 352.459,A -85,B 0,C 180,E1 -9900,E2 -9900} C_VEL
LIN {X 0,Y 425.551,Z 352.476,A -85,B 0,C 180,E1 -9902.84,E2 -9902.84} C_VEL
LIN {X 0,Y 425.536,Z 352.478,A -85,B 0,C 180,E1 -9906.651,E2 -9906.651} C_VEL
LIN {X 0,Y 425.408,Z 352.495,A -85,B 0,C 180,E1 -9909.509,E2 -9909.509} C_VEL
LIN {X 0,Y 425.4,Z 352.494,A -85,B 0,C 180,E1 -9912.904,E2 -9912.904} C_VEL
LIN {X 0,Y 425.368,Z 352.499,A -85,B 0,C 180,E1 -9916.605,E2 -9916.605} C_VEL
LIN {X 0,Y 425.335,Z 352.505,A -85,B 0,C 180,E1 -9919.636,E2 -9919.636} C_VEL
LIN {X 0,Y 425.314,Z 352.507,A -85,B 0,C 180,E1 -9923.365,E2 -9923.365} C_VEL
LIN {X 0,Y 425.353,Z 352.5,A -85,B 0,C 180,E1 -9926.844,E2 -9926.844} C_VEL
LIN {X 0,Y 425.297,Z 352.511,A -85,B 0,C 180,E1 -9929.719,E2 -9929.719} C_VEL
LIN {X 0,Y 425.289,Z 352.51,A -85,B 0,C 180,E1 -9933.048,E2 -9933.048} C_VEL
LIN {X 0,Y 425.288,Z 352.51,A -85,B 0,C 180,E1 -9935.929,E2 -9935.929} C_VEL
LIN {X 0,Y 425.304,Z 352.508,A -85,B 0,C 180,E1 -9939.043,E2 -9939.043} C_VEL
LIN {X 0,Y 425.281,Z 352.51,A -85,B 0,C 180,E1 -9942.653,E2 -9942.653} C_VEL
LIN {X 0,Y 425.268,Z 352.511,A -85,B 0,C 180,E1 -9946.044,E2 -9946.044} C_VEL
LIN {X 0,Y 425.281,Z 352.51,A -85,B 0,C 180,E1 -9948.621,E2 -9948.621} C_VEL
LIN {X 0,Y 425.312,Z 352.509,A -85,B 0,C 180,E1 -9951.102,E2 -9951.102} C_VEL
LIN {X 0,Y 425.305,Z 352.507,A -85,B 0,C 180,E1 -9954.664,E2 -9954.664} C_VEL
LIN {X 0,Y 425.271,Z 352.51,A -85,B 0,C 180,E1 -9958.073,E2 -9958.073} C_VEL
LIN {X 0,Y 425.338,Z 352.505,A -85,B 0,C 180,E1 -9961.368,E2 -9961.368} C_VEL
LIN {X 0,Y 425.302,Z 352.509,A -85,B 0,C 180,E1 -9964.554,E2 -9964.554} C_VEL
LIN {X 0,Y 425.294,Z 352.507,A -85,B 0,C 180,E1 -9967.661,E2 -9967.661} C_VEL
LIN {X 0,Y 425.369,Z 352.502,A -85,B 0,C 180,E1 -9970.704,E2 -9970.704} C_VEL
LIN {X 0,Y 425.395,Z 352.495,A -85,B 0,C 180,E1 -9973.688,E2 -9973.688} C_VEL
LIN {X 0,Y 425.419,Z 352.492,A -85,B 0,C 180,E1 -9977.598,E2 -9977.598} C_VEL
LIN {X 0,Y 425.48,Z 352.487,A -85,B 0,C 180,E1 -9981.685,E2 -9981.685} C_VEL
LIN {X 0,Y 425.483,Z 352.487,A -85,B 0,C 180,E1 -9981.781,E2 -9981.781} C_VEL
LIN {X 0,Y 428.736,Z 364.038,A -85,B 0,C 180,E1 -9982.464,E2 -9982.464} C_VEL
LIN {X 0,Y 429.219,Z 366.012,A -85,B 0,C 180,E1 -9982.591,E2 -9982.591} C_VEL
LIN {X 0,Y 428.777,Z 378.42,A -85,B 0,C 180,E1 -9983.411,E2 -9983.411} C_VEL
LIN {X 0,Y 428.158,Z 389.493,A -85,B 0,C 180,E1 -9984.347,E2 -9984.347} C_VEL
LIN {X 0,Y 427.649,Z 398.44,A -85,B 0,C 180,E1 -9985.286,E2 -9985.286} C_VEL
LIN {X 0,Y 427.072,Z 407.651,A -85,B 0,C 180,E1 -9986.461,E2 -9986.461} C_VEL
LIN {X 0,Y 426.467,Z 416.533,A -85,B 0,C 180,E1 -9987.874,E2 -9987.874} C_VEL
LIN {X 0,Y 425.91,Z 423.709,A -85,B 0,C 180,E1 -9989.29,E2 -9989.29} C_VEL
LIN {X 0,Y 425.609,Z 428.565,A -85,B 0,C 180,E1 -9990.472,E2 -9990.472} C_VEL
LIN {X 0,Y 425.394,Z 433.275,A -85,B 0,C 180,E1 -9991.893,E2 -9991.893} C_VEL
LIN {X 0,Y 425.196,Z 435.313,A -85,B 0,C 180,E1 -9992.634,E2 -9992.634} C_VEL
LIN {X 0,Y 424.392,Z 437.189,A -85,B 0,C 180,E1 -9993.383,E2 -9993.383} C_VEL
LIN {X 0,Y 421.419,Z 439.838,A -85,B 0,C 180,E1 -9994.614,E2 -9994.614} C_VEL
LIN {X 0,Y 418.979,Z 441.483,A -85,B 0,C 180,E1 -9995.623,E2 -9995.623} C_VEL
LIN {X 0,Y 417.938,Z 442.353,A -85,B 0,C 180,E1 -9996.412,E2 -9996.412} C_VEL
LIN {X 0,Y 417.853,Z 442.557,A -85,B 0,C 180,E1 -9996.681,E2 -9996.681} C_VEL
LIN {X 0,Y 417.876,Z 443.019,A -85,B 0,C 180,E1 -9997.732,E2 -9997.732} C_VEL
LIN {X 0,Y 417.857,Z 442.699,A -85,B 0,C 180,E1 -9999.682,E2 -9999.682} C_VEL
LIN {X 0,Y 417.929,Z 441.933,A -85,B 0,C 180,E1 -10000.659,E2 -10000.659} C_VEL
LIN {X 0,Y 418.245,Z 439.143,A -85,B 0,C 180,E1 -10002.617,E2 -10002.617} C_VEL
LIN {X 0,Y 418.496,Z 435.917,A -85,B 0,C 180,E1 -10004.093,E2 -10004.093} C_VEL
LIN {X 0,Y 418.894,Z 431.592,A -85,B 0,C 180,E1 -10005.571,E2 -10005.571} C_VEL
LIN {X 0,Y 419.466,Z 425.194,A -85,B 0,C 180,E1 -10007.249,E2 -10007.249} C_VEL
LIN {X 0,Y 420.086,Z 417.667,A -85,B 0,C 180,E1 -10008.786,E2 -10008.786} C_VEL
LIN {X 0,Y 420.745,Z 410.169,A -85,B 0,C 180,E1 -10010.024,E2 -10010.024} C_VEL
LIN {X 0,Y 421.457,Z 400.691,A -85,B 0,C 180,E1 -10011.307,E2 -10011.307} C_VEL
LIN {X 0,Y 422.19,Z 390.757,A -85,B 0,C 180,E1 -10012.382,E2 -10012.382} C_VEL
LIN {X 0,Y 422.753,Z 380.858,A -85,B 0,C 180,E1 -10013.254,E2 -10013.254} C_VEL
LIN {X 0,Y 423.387,Z 368.939,A -85,B 0,C 180,E1 -10014.079,E2 -10014.079} C_VEL
LIN {X 0,Y 419.468,Z 357.127,A -85,B 0,C 180,E1 -10014.927,E2 -10014.927} C_VEL
LIN {X 0,Y 418.27,Z 353.386,A -85,B 0,C 180,E1 -10015.149,E2 -10015.149} C_VEL
LIN {X 0,Y 418.293,Z 353.384,A -85,B 0,C 180,E1 -10018.062,E2 -10018.062} C_VEL
LIN {X 0,Y 418.213,Z 353.393,A -85,B 0,C 180,E1 -10021.395,E2 -10021.395} C_VEL
LIN {X 0,Y 418.266,Z 353.387,A -85,B 0,C 180,E1 -10024.579,E2 -10024.579} C_VEL
LIN {X 0,Y 418.229,Z 353.39,A -85,B 0,C 180,E1 -10027.833,E2 -10027.833} C_VEL
LIN {X 0,Y 418.223,Z 353.391,A -85,B 0,C 180,E1 -10030.947,E2 -10030.947} C_VEL
LIN {X 0,Y 418.216,Z 353.392,A -85,B 0,C 180,E1 -10033.73,E2 -10033.73} C_VEL
LIN {X 0,Y 418.208,Z 353.393,A -85,B 0,C 180,E1 -10036.448,E2 -10036.448} C_VEL
LIN {X 0,Y 418.264,Z 353.388,A -85,B 0,C 180,E1 -10039.123,E2 -10039.123} C_VEL
LIN {X 0,Y 418.238,Z 353.391,A -85,B 0,C 180,E1 -10042.164,E2 -10042.164} C_VEL
LIN {X 0,Y 418.264,Z 353.387,A -85,B 0,C 180,E1 -10045.419,E2 -10045.419} C_VEL
LIN {X 0,Y 418.219,Z 353.378,A -85,B 0,C 180,E1 -10048.604,E2 -10048.604} C_VEL
LIN {X 0,Y 418.293,Z 353.374,A -85,B 0,C 180,E1 -10051.936,E2 -10051.936} C_VEL
LIN {X 0,Y 418.287,Z 353.382,A -85,B 0,C 180,E1 -10055.162,E2 -10055.162} C_VEL
LIN {X 0,Y 418.232,Z 353.387,A -85,B 0,C 180,E1 -10058.303,E2 -10058.303} C_VEL
LIN {X 0,Y 418.281,Z 353.379,A -85,B 0,C 180,E1 -10061.383,E2 -10061.383} C_VEL
LIN {X 0,Y 418.3,Z 353.382,A -85,B 0,C 180,E1 -10064.406,E2 -10064.406} C_VEL
LIN {X 0,Y 418.368,Z 353.373,A -85,B 0,C 180,E1 -10067.386,E2 -10067.386} C_VEL
LIN {X 0,Y 418.358,Z 353.373,A -85,B 0,C 180,E1 -10070.329,E2 -10070.329} C_VEL
LIN {X 0,Y 418.491,Z 353.354,A -85,B 0,C 180,E1 -10073.249,E2 -10073.249} C_VEL
LIN {X 0,Y 418.339,Z 353.371,A -85,B 0,C 180,E1 -10075.181,E2 -10075.181} C_VEL
LIN {X 0,Y 418.542,Z 353.351,A -85,B 0,C 180,E1 -10078.075,E2 -10078.075} C_VEL
LIN {X 0,Y 418.671,Z 353.328,A -85,B 0,C 180,E1 -10080,E2 -10080} C_VEL
LIN {X 0,Y 418.508,Z 353.356,A -85,B 0,C 180,E1 -10082.888,E2 -10082.888} C_VEL
LIN {X 0,Y 418.49,Z 353.357,A -85,B 0,C 180,E1 -10086.751,E2 -10086.751} C_VEL
LIN {X 0,Y 418.338,Z 353.371,A -85,B 0,C 180,E1 -10089.671,E2 -10089.671} C_VEL
LIN {X 0,Y 418.342,Z 353.375,A -85,B 0,C 180,E1 -10093.001,E2 -10093.001} C_VEL
LIN {X 0,Y 418.309,Z 353.379,A -85,B 0,C 180,E1 -10096.736,E2 -10096.736} C_VEL
LIN {X 0,Y 418.267,Z 353.386,A -85,B 0,C 180,E1 -10099.791,E2 -10099.791} C_VEL
LIN {X 0,Y 418.234,Z 353.39,A -85,B 0,C 180,E1 -10102.736,E2 -10102.736} C_VEL
LIN {X 0,Y 418.267,Z 353.387,A -85,B 0,C 180,E1 -10105.904,E2 -10105.904} C_VEL
LIN {X 0,Y 418.271,Z 353.388,A -85,B 0,C 180,E1 -10109.161,E2 -10109.161} C_VEL
LIN {X 0,Y 418.254,Z 353.388,A -85,B 0,C 180,E1 -10112.844,E2 -10112.844} C_VEL
LIN {X 0,Y 418.246,Z 353.388,A -85,B 0,C 180,E1 -10116.239,E2 -10116.239} C_VEL
LIN {X 0,Y 418.264,Z 353.386,A -85,B 0,C 180,E1 -10119.681,E2 -10119.681} C_VEL
LIN {X 0,Y 418.282,Z 353.38,A -85,B 0,C 180,E1 -10122.33,E2 -10122.33} C_VEL
LIN {X 0,Y 418.272,Z 353.385,A -85,B 0,C 180,E1 -10125.115,E2 -10125.115} C_VEL
LIN {X 0,Y 418.314,Z 353.51,A -85,B 0,C 180,E1 -10126.935,E2 -10126.935} C_VEL
LIN {X 0,Y 419.843,Z 361.027,A -85,B 0,C 180,E1 -10129.833,E2 -10129.833} C_VEL
LIN {X 0,Y 421.181,Z 368.335,A -85,B 0,C 180,E1 -10132.48,E2 -10132.48} C_VEL
LIN {X 0,Y 421.404,Z 372.039,A -85,B 0,C 180,E1 -10133.734,E2 -10133.734} C_VEL
LIN {X 0,Y 420.265,Z 384.424,A -85,B 0,C 180,E1 -10137.648,E2 -10137.648} C_VEL
LIN {X 0,Y 419.498,Z 395.229,A -85,B 0,C 180,E1 -10140.933,E2 -10140.933} C_VEL
LIN {X 0,Y 418.875,Z 406.043,A -85,B 0,C 180,E1 -10144.137,E2 -10144.137} C_VEL
LIN {X 0,Y 418.331,Z 417.721,A -85,B 0,C 180,E1 -10147.519,E2 -10147.519} C_VEL
LIN {X 0,Y 417.871,Z 429.415,A -85,B 0,C 180,E1 -10150.856,E2 -10150.856} C_VEL
LIN {X 0,Y 417.73,Z 435.082,A -85,B 0,C 180,E1 -10152.428,E2 -10152.428} C_VEL
LIN {X 0,Y 419.707,Z 449.198,A -85,B 0,C 180,E1 -10152.911,E2 -10152.911} C_VEL
LIN {X 0,Y 420.719,Z 461.798,A -85,B 0,C 180,E1 -10153.503,E2 -10153.503} C_VEL
LIN {X 0,Y 421.232,Z 472.417,A -85,B 0,C 180,E1 -10154.146,E2 -10154.146} C_VEL
LIN {X 0,Y 420.376,Z 483.931,A -85,B 0,C 180,E1 -10154.982,E2 -10154.982} C_VEL
LIN {X 0,Y 419.525,Z 495.639,A -85,B 0,C 180,E1 -10156.066,E2 -10156.066} C_VEL
LIN {X 0,Y 418.965,Z 505.395,A -85,B 0,C 180,E1 -10157.191,E2 -10157.191} C_VEL
LIN {X 0,Y 418.316,Z 513.823,A -85,B 0,C 180,E1 -10158.37,E2 -10158.37} C_VEL
LIN {X 0,Y 417.731,Z 522.307,A -85,B 0,C 180,E1 -10159.826,E2 -10159.826} C_VEL
LIN {X 0,Y 417.527,Z 529.201,A -85,B 0,C 180,E1 -10161.287,E2 -10161.287} C_VEL
LIN {X 0,Y 417.367,Z 534.734,A -85,B 0,C 180,E1 -10162.745,E2 -10162.745} C_VEL
LIN {X 0,Y 417.424,Z 539.092,A -85,B 0,C 180,E1 -10164.203,E2 -10164.203} C_VEL
LIN {X 0,Y 417.382,Z 541.405,A -85,B 0,C 180,E1 -10165.171,E2 -10165.171} C_VEL
LIN {X 0,Y 417.505,Z 543.251,A -85,B 0,C 180,E1 -10166.14,E2 -10166.14} C_VEL
LIN {X 0,Y 417.519,Z 544.649,A -85,B 0,C 180,E1 -10167.106,E2 -10167.106} C_VEL
LIN {X 0,Y 417.483,Z 546.231,A -85,B 0,C 180,E1 -10169.036,E2 -10169.036} C_VEL
LIN {X 0,Y 417.516,Z 546.387,A -85,B 0,C 180,E1 -10170.001,E2 -10170.001} C_VEL
LIN {X 0,Y 417.496,Z 546.124,A -85,B 0,C 180,E1 -10170.965,E2 -10170.965} C_VEL
LIN {X 0,Y 417.494,Z 545.465,A -85,B 0,C 180,E1 -10171.93,E2 -10171.93} C_VEL
LIN {X 0,Y 417.528,Z 544.41,A -85,B 0,C 180,E1 -10172.895,E2 -10172.895} C_VEL
LIN {X 0,Y 417.571,Z 542.895,A -85,B 0,C 180,E1 -10173.861,E2 -10173.861} C_VEL
LIN {X 0,Y 417.405,Z 539.77,A -85,B 0,C 180,E1 -10175.314,E2 -10175.314} C_VEL
LIN {X 0,Y 417.439,Z 535.577,A -85,B 0,C 180,E1 -10176.769,E2 -10176.769} C_VEL
LIN {X 0,Y 417.523,Z 529.141,A -85,B 0,C 180,E1 -10178.47,E2 -10178.47} C_VEL
LIN {X 0,Y 417.694,Z 522.137,A -85,B 0,C 180,E1 -10179.932,E2 -10179.932} C_VEL
LIN {X 0,Y 418.183,Z 513.435,A -85,B 0,C 180,E1 -10181.39,E2 -10181.39} C_VEL
LIN {X 0,Y 418.763,Z 504.505,A -85,B 0,C 180,E1 -10182.603,E2 -10182.603} C_VEL
LIN {X 0,Y 419.353,Z 493.505,A -85,B 0,C 180,E1 -10183.817,E2 -10183.817} C_VEL
LIN {X 0,Y 420.021,Z 482.508,A -85,B 0,C 180,E1 -10184.784,E2 -10184.784} C_VEL
LIN {X 0,Y 420.729,Z 470.23,A -85,B 0,C 180,E1 -10185.624,E2 -10185.624} C_VEL
LIN {X 0,Y 419.782,Z 457.314,A -85,B 0,C 180,E1 -10186.33,E2 -10186.33} C_VEL
LIN {X 0,Y 418.553,Z 444.28,A -85,B 0,C 180,E1 -10186.843,E2 -10186.843} C_VEL
LIN {X 0,Y 417.671,Z 435.489,A -85,B 0,C 180,E1 -10187.11,E2 -10187.11} C_VEL
LIN {X 0,Y 418.009,Z 422.683,A -85,B 0,C 180,E1 -10190.676,E2 -10190.676} C_VEL
LIN {X 0,Y 418.488,Z 409.806,A -85,B 0,C 180,E1 -10194.297,E2 -10194.297} C_VEL
LIN {X 0,Y 419.088,Z 396.798,A -85,B 0,C 180,E1 -10198.006,E2 -10198.006} C_VEL
LIN {X 0,Y 419.719,Z 385.313,A -85,B 0,C 180,E1 -10201.354,E2 -10201.354} C_VEL
LIN {X 0,Y 420.515,Z 373.079,A -85,B 0,C 180,E1 -10205.022,E2 -10205.022} C_VEL
LIN {X 0,Y 420.792,Z 367.616,A -85,B 0,C 180,E1 -10206.708,E2 -10206.708} C_VEL
LIN {X 0,Y 419.36,Z 359.078,A -85,B 0,C 180,E1 -10209.564,E2 -10209.564} C_VEL
LIN {X 0,Y 418.283,Z 353.384,A -85,B 0,C 180,E1 -10211.581,E2 -10211.581} C_VEL
LIN {X 0,Y 418.242,Z 353.39,A -85,B 0,C 180,E1 -10215.11,E2 -10215.11} C_VEL
LIN {X 0,Y 418.244,Z 353.386,A -85,B 0,C 180,E1 -10217.767,E2 -10217.767} C_VEL
LIN {X 0,Y 418.26,Z 353.386,A -85,B 0,C 180,E1 -10220.619,E2 -10220.619} C_VEL
LIN {X 0,Y 418.247,Z 353.385,A -85,B 0,C 180,E1 -10223.976,E2 -10223.976} C_VEL
LIN {X 0,Y 418.262,Z 353.386,A -85,B 0,C 180,E1 -10227.156,E2 -10227.156} C_VEL
LIN {X 0,Y 418.273,Z 353.386,A -85,B 0,C 180,E1 -10230.896,E2 -10230.896} C_VEL
LIN {X 0,Y 418.276,Z 353.382,A -85,B 0,C 180,E1 -10234.096,E2 -10234.096} C_VEL
LIN {X 0,Y 418.243,Z 353.387,A -85,B 0,C 180,E1 -10237.264,E2 -10237.264} C_VEL
LIN {X 0,Y 418.288,Z 353.383,A -85,B 0,C 180,E1 -10240.365,E2 -10240.365} C_VEL
LIN {X 0,Y 418.322,Z 353.375,A -85,B 0,C 180,E1 -10243.405,E2 -10243.405} C_VEL
LIN {X 0,Y 418.352,Z 353.374,A -85,B 0,C 180,E1 -10247,E2 -10247} C_VEL
LIN {X 0,Y 418.346,Z 353.377,A -85,B 0,C 180,E1 -10250.329,E2 -10250.329} C_VEL
LIN {X 0,Y 418.519,Z 353.355,A -85,B 0,C 180,E1 -10252.28,E2 -10252.28} C_VEL
LIN {X 0,Y 418.519,Z 353.355,A -85,B 0,C 180,E1 -10254.218,E2 -10254.218} C_VEL
LIN {X 0,Y 418.548,Z 353.351,A -85,B 0,C 180,E1 -10258.076,E2 -10258.076} C_VEL
LIN {X 0,Y 418.679,Z 353.335,A -85,B 0,C 180,E1 -10260,E2 -10260} C_VEL
LIN {X 0,Y 418.506,Z 353.353,A -85,B 0,C 180,E1 -10262.888,E2 -10262.888} C_VEL
LIN {X 0,Y 418.5,Z 353.354,A -85,B 0,C 180,E1 -10266.751,E2 -10266.751} C_VEL
LIN {X 0,Y 418.407,Z 353.366,A -85,B 0,C 180,E1 -10268.695,E2 -10268.695} C_VEL
LIN {X 0,Y 418.322,Z 353.379,A -85,B 0,C 180,E1 -10271.631,E2 -10271.631} C_VEL
LIN {X 0,Y 418.309,Z 353.378,A -85,B 0,C 180,E1 -10274.597,E2 -10274.597} C_VEL
LIN {X 0,Y 418.295,Z 353.382,A -85,B 0,C 180,E1 -10277.604,E2 -10277.604} C_VEL
LIN {X 0,Y 418.256,Z 353.384,A -85,B 0,C 180,E1 -10280.663,E2 -10280.663} C_VEL
LIN {X 0,Y 418.295,Z 353.383,A -85,B 0,C 180,E1 -10283.781,E2 -10283.781} C_VEL
LIN {X 0,Y 418.316,Z 353.378,A -85,B 0,C 180,E1 -10287.07,E2 -10287.07} C_VEL
LIN {X 0,Y 418.251,Z 353.385,A -85,B 0,C 180,E1 -10290.272,E2 -10290.272} C_VEL
LIN {X 0,Y 418.255,Z 353.388,A -85,B 0,C 180,E1 -10293.677,E2 -10293.677} C_VEL
LIN {X 0,Y 418.247,Z 353.389,A -85,B 0,C 180,E1 -10297.224,E2 -10297.224} C_VEL
LIN {X 0,Y 418.258,Z 353.387,A -85,B 0,C 180,E1 -10299.682,E2 -10299.682} C_VEL
LIN {X 0,Y 418.236,Z 353.387,A -85,B 0,C 180,E1 -10302.321,E2 -10302.321} C_VEL
LIN {X 0,Y 418.242,Z 353.39,A -85,B 0,C 180,E1 -10305.109,E2 -10305.109} C_VEL
LIN {X 0,Y 418.246,Z 353.387,A -85,B 0,C 180,E1 -10307.767,E2 -10307.767} C_VEL
LIN {X 0,Y 418.259,Z 353.385,A -85,B 0,C 180,E1 -10310.619,E2 -10310.619} C_VEL
LIN {X 0,Y 418.248,Z 353.385,A -85,B 0,C 180,E1 -10313.975,E2 -10313.975} C_VEL
LIN {X 0,Y 418.264,Z 353.387,A -85,B 0,C 180,E1 -10317.156,E2 -10317.156} C_VEL
LIN {X 0,Y 418.275,Z 353.385,A -85,B 0,C 180,E1 -10320.895,E2 -10320.895} C_VEL
LIN {X 0,Y 418.277,Z 353.382,A -85,B 0,C 180,E1 -10324.096,E2 -10324.096} C_VEL
LIN {X 0,Y 418.245,Z 353.388,A -85,B 0,C 180,E1 -10327.263,E2 -10327.263} C_VEL
LIN {X 0,Y 418.29,Z 353.381,A -85,B 0,C 180,E1 -10330.364,E2 -10330.364} C_VEL
LIN {X 0,Y 418.324,Z 353.377,A -85,B 0,C 180,E1 -10333.404,E2 -10333.404} C_VEL
LIN {X 0,Y 418.353,Z 353.376,A -85,B 0,C 180,E1 -10336.999,E2 -10336.999} C_VEL
LIN {X 0,Y 418.348,Z 353.375,A -85,B 0,C 180,E1 -10340.328,E2 -10340.328} C_VEL
LIN {X 0,Y 418.454,Z 353.476,A -85,B 0,C 180,E1 -10341.552,E2 -10341.552} C_VEL
LIN {X 0,Y 421.768,Z 365.068,A -85,B 0,C 180,E1 -10342.245,E2 -10342.245} C_VEL
LIN {X 0,Y 422.333,Z 368.505,A -85,B 0,C 180,E1 -10342.469,E2 -10342.469} C_VEL
LIN {X 0,Y 421.819,Z 380.59,A -85,B 0,C 180,E1 -10343.302,E2 -10343.302} C_VEL
LIN {X 0,Y 421.231,Z 391.398,A -85,B 0,C 180,E1 -10344.254,E2 -10344.254} C_VEL
LIN {X 0,Y 420.698,Z 400.169,A -85,B 0,C 180,E1 -10345.208,E2 -10345.208} C_VEL
LIN {X 0,Y 420.082,Z 409.187,A -85,B 0,C 180,E1 -10346.402,E2 -10346.402} C_VEL
LIN {X 0,Y 419.478,Z 417.952,A -85,B 0,C 180,E1 -10347.839,E2 -10347.839} C_VEL
LIN {X 0,Y 418.907,Z 425.034,A -85,B 0,C 180,E1 -10349.278,E2 -10349.278} C_VEL
LIN {X 0,Y 418.584,Z 429.806,A -85,B 0,C 180,E1 -10350.48,E2 -10350.48} C_VEL
LIN {X 0,Y 418.342,Z 434.441,A -85,B 0,C 180,E1 -10351.925,E2 -10351.925} C_VEL
LIN {X 0,Y 418.026,Z 438.022,A -85,B 0,C 180,E1 -10353.373,E2 -10353.373} C_VEL
LIN {X 0,Y 417.966,Z 440.588,A -85,B 0,C 180,E1 -10354.822,E2 -10354.822} C_VEL
LIN {X 0,Y 417.915,Z 441.808,A -85,B 0,C 180,E1 -10355.79,E2 -10355.79} C_VEL
LIN {X 0,Y 417.853,Z 442.557,A -85,B 0,C 180,E1 -10356.681,E2 -10356.681} C_VEL
LIN {X 0,Y 417.182,Z 443.161,A -85,B 0,C 180,E1 -10357.482,E2 -10357.482} C_VEL
LIN {X 0,Y 414.329,Z 443.692,A -85,B 0,C 180,E1 -10358.791,E2 -10358.791} C_VEL
LIN {X 0,Y 411.513,Z 443.353,A -85,B 0,C 180,E1 -10360.114,E2 -10360.114} C_VEL
LIN {X 0,Y 410.913,Z 442.591,A -85,B 0,C 180,E1 -10360.928,E2 -10360.928} C_VEL
LIN {X 0,Y 411.257,Z 439.839,A -85,B 0,C 180,E1 -10362.835,E2 -10362.835} C_VEL
LIN {X 0,Y 411.549,Z 436.54,A -85,B 0,C 180,E1 -10364.336,E2 -10364.336} C_VEL
LIN {X 0,Y 411.97,Z 432.14,A -85,B 0,C 180,E1 -10365.839,E2 -10365.839} C_VEL
LIN {X 0,Y 412.549,Z 426.058,A -85,B 0,C 180,E1 -10367.446,E2 -10367.446} C_VEL
LIN {X 0,Y 413.138,Z 419.342,A -85,B 0,C 180,E1 -10368.857,E2 -10368.857} C_VEL
LIN {X 0,Y 413.983,Z 410.378,A -85,B 0,C 180,E1 -10370.365,E2 -10370.365} C_VEL
LIN {X 0,Y 414.717,Z 400.894,A -85,B 0,C 180,E1 -10371.647,E2 -10371.647} C_VEL
LIN {X 0,Y 415.468,Z 390.569,A -85,B 0,C 180,E1 -10372.764,E2 -10372.764} C_VEL
LIN {X 0,Y 416.155,Z 380.434,A -85,B 0,C 180,E1 -10373.645,E2 -10373.645} C_VEL
LIN {X 0,Y 416.6,Z 370.281,A -85,B 0,C 180,E1 -10374.358,E2 -10374.358} C_VEL
LIN {X 0,Y 412.9,Z 359.236,A -85,B 0,C 180,E1 -10375.183,E2 -10375.183} C_VEL
LIN {X 0,Y 411.25,Z 354.26,A -85,B 0,C 180,E1 -10375.505,E2 -10375.505} C_VEL
LIN {X 0,Y 411.22,Z 354.264,A -85,B 0,C 180,E1 -10378.589,E2 -10378.589} C_VEL
LIN {X 0,Y 411.167,Z 354.274,A -85,B 0,C 180,E1 -10381.996,E2 -10381.996} C_VEL
LIN {X 0,Y 411.211,Z 354.267,A -85,B 0,C 180,E1 -10384.878,E2 -10384.878} C_VEL
LIN {X 0,Y 411.206,Z 354.264,A -85,B 0,C 180,E1 -10388.168,E2 -10388.168} C_VEL
LIN {X 0,Y 411.165,Z 354.271,A -85,B 0,C 180,E1 -10391.228,E2 -10391.228} C_VEL
LIN {X 0,Y 411.179,Z 354.268,A -85,B 0,C 180,E1 -10394.489,E2 -10394.489} C_VEL
LIN {X 0,Y 411.198,Z 354.268,A -85,B 0,C 180,E1 -10398.197,E2 -10398.197} C_VEL
LIN {X 0,Y 411.231,Z 354.263,A -85,B 0,C 180,E1 -10400.777,E2 -10400.777} C_VEL
LIN {X 0,Y 411.198,Z 354.265,A -85,B 0,C 180,E1 -10404.471,E2 -10404.471} C_VEL
LIN {X 0,Y 411.169,Z 354.261,A -85,B 0,C 180,E1 -10408.003,E2 -10408.003} C_VEL
LIN {X 0,Y 411.222,Z 354.249,A -85,B 0,C 180,E1 -10411.41,E2 -10411.41} C_VEL
LIN {X 0,Y 411.234,Z 354.26,A -85,B 0,C 180,E1 -10414.706,E2 -10414.706} C_VEL
LIN {X 0,Y 411.203,Z 354.261,A -85,B 0,C 180,E1 -10417.913,E2 -10417.913} C_VEL
LIN {X 0,Y 411.222,Z 354.261,A -85,B 0,C 180,E1 -10421.051,E2 -10421.051} C_VEL
LIN {X 0,Y 411.252,Z 354.258,A -85,B 0,C 180,E1 -10424.131,E2 -10424.131} C_VEL
LIN {X 0,Y 411.312,Z 354.25,A -85,B 0,C 180,E1 -10427.166,E2 -10427.166} C_VEL
LIN {X 0,Y 411.307,Z 354.25,A -85,B 0,C 180,E1 -10430.161,E2 -10430.161} C_VEL
LIN {X 0,Y 411.457,Z 354.231,A -85,B 0,C 180,E1 -10433.133,E2 -10433.133} C_VEL
LIN {X 0,Y 411.31,Z 354.246,A -85,B 0,C 180,E1 -10435.099,E2 -10435.099} C_VEL
LIN {X 0,Y 411.511,Z 354.227,A -85,B 0,C 180,E1 -10438.042,E2 -10438.042} C_VEL
LIN {X 0,Y 411.641,Z 354.203,A -85,B 0,C 180,E1 -10440,E2 -10440} C_VEL
LIN {X 0,Y 411.463,Z 354.233,A -85,B 0,C 180,E1 -10442.937,E2 -10442.937} C_VEL
LIN {X 0,Y 411.457,Z 354.233,A -85,B 0,C 180,E1 -10446.867,E2 -10446.867} C_VEL
LIN {X 0,Y 411.289,Z 354.248,A -85,B 0,C 180,E1 -10449.839,E2 -10449.839} C_VEL
LIN {X 0,Y 411.301,Z 354.251,A -85,B 0,C 180,E1 -10453.104,E2 -10453.104} C_VEL
LIN {X 0,Y 411.259,Z 354.257,A -85,B 0,C 180,E1 -10456.869,E2 -10456.869} C_VEL
LIN {X 0,Y 411.226,Z 354.263,A -85,B 0,C 180,E1 -10459.987,E2 -10459.987} C_VEL
LIN {X 0,Y 411.199,Z 354.266,A -85,B 0,C 180,E1 -10463.148,E2 -10463.148} C_VEL
LIN {X 0,Y 411.234,Z 354.265,A -85,B 0,C 180,E1 -10466.381,E2 -10466.381} C_VEL
LIN {X 0,Y 411.207,Z 354.266,A -85,B 0,C 180,E1 -10469.712,E2 -10469.712} C_VEL
LIN {X 0,Y 411.203,Z 354.267,A -85,B 0,C 180,E1 -10473.156,E2 -10473.156} C_VEL
LIN {X 0,Y 411.193,Z 354.268,A -85,B 0,C 180,E1 -10476.554,E2 -10476.554} C_VEL
LIN {X 0,Y 411.226,Z 354.262,A -85,B 0,C 180,E1 -10479.731,E2 -10479.731} C_VEL
LIN {X 0,Y 411.225,Z 354.264,A -85,B 0,C 180,E1 -10483.127,E2 -10483.127} C_VEL
LIN {X 0,Y 411.232,Z 354.302,A -85,B 0,C 180,E1 -10486.5,E2 -10486.5} C_VEL
LIN {X 0,Y 413.037,Z 363.14,A -85,B 0,C 180,E1 -10489.969,E2 -10489.969} C_VEL
LIN {X 0,Y 414.401,Z 371.02,A -85,B 0,C 180,E1 -10492.853,E2 -10492.853} C_VEL
LIN {X 0,Y 414.309,Z 374.81,A -85,B 0,C 180,E1 -10494.128,E2 -10494.128} C_VEL
LIN {X 0,Y 413.279,Z 385.661,A -85,B 0,C 180,E1 -10497.611,E2 -10497.611} C_VEL
LIN {X 0,Y 412.453,Z 396.41,A -85,B 0,C 180,E1 -10500.947,E2 -10500.947} C_VEL
LIN {X 0,Y 411.814,Z 407.192,A -85,B 0,C 180,E1 -10504.204,E2 -10504.204} C_VEL
LIN {X 0,Y 411.215,Z 419.752,A -85,B 0,C 180,E1 -10507.915,E2 -10507.915} C_VEL
LIN {X 0,Y 410.715,Z 432.228,A -85,B 0,C 180,E1 -10511.545,E2 -10511.545} C_VEL
LIN {X 0,Y 410.662,Z 434.077,A -85,B 0,C 180,E1 -10512.071,E2 -10512.071} C_VEL
LIN {X 0,Y 412.673,Z 448.117,A -85,B 0,C 180,E1 -10512.564,E2 -10512.564} C_VEL
LIN {X 0,Y 413.749,Z 460.106,A -85,B 0,C 180,E1 -10513.137,E2 -10513.137} C_VEL
LIN {X 0,Y 414.326,Z 472.066,A -85,B 0,C 180,E1 -10513.874,E2 -10513.874} C_VEL
LIN {X 0,Y 413.506,Z 483.464,A -85,B 0,C 180,E1 -10514.726,E2 -10514.726} C_VEL
LIN {X 0,Y 412.591,Z 495.091,A -85,B 0,C 180,E1 -10515.827,E2 -10515.827} C_VEL
LIN {X 0,Y 411.995,Z 504.996,A -85,B 0,C 180,E1 -10517,E2 -10517} C_VEL
LIN {X 0,Y 411.294,Z 513.147,A -85,B 0,C 180,E1 -10518.168,E2 -10518.168} C_VEL
LIN {X 0,Y 410.694,Z 521.589,A -85,B 0,C 180,E1 -10519.65,E2 -10519.65} C_VEL
LIN {X 0,Y 410.446,Z 528.449,A -85,B 0,C 180,E1 -10521.136,E2 -10521.136} C_VEL
LIN {X 0,Y 410.293,Z 533.956,A -85,B 0,C 180,E1 -10522.62,E2 -10522.62} C_VEL
LIN {X 0,Y 410.336,Z 538.29,A -85,B 0,C 180,E1 -10524.102,E2 -10524.102} C_VEL
LIN {X 0,Y 410.304,Z 540.59,A -85,B 0,C 180,E1 -10525.088,E2 -10525.088} C_VEL
LIN {X 0,Y 410.436,Z 542.418,A -85,B 0,C 180,E1 -10526.073,E2 -10526.073} C_VEL
LIN {X 0,Y 410.47,Z 543.81,A -85,B 0,C 180,E1 -10527.056,E2 -10527.056} C_VEL
LIN {X 0,Y 410.433,Z 545.369,A -85,B 0,C 180,E1 -10529.02,E2 -10529.02} C_VEL
LIN {X 0,Y 410.471,Z 545.509,A -85,B 0,C 180,E1 -10530.001,E2 -10530.001} C_VEL
LIN {X 0,Y 410.449,Z 545.236,A -85,B 0,C 180,E1 -10530.982,E2 -10530.982} C_VEL
LIN {X 0,Y 410.445,Z 544.567,A -85,B 0,C 180,E1 -10531.963,E2 -10531.963} C_VEL
LIN {X 0,Y 410.482,Z 543.499,A -85,B 0,C 180,E1 -10532.945,E2 -10532.945} C_VEL
LIN {X 0,Y 410.435,Z 541.033,A -85,B 0,C 180,E1 -10534.42,E2 -10534.42} C_VEL
LIN {X 0,Y 410.39,Z 537.537,A -85,B 0,C 180,E1 -10535.898,E2 -10535.898} C_VEL
LIN {X 0,Y 410.37,Z 532.925,A -85,B 0,C 180,E1 -10537.38,E2 -10537.38} C_VEL
LIN {X 0,Y 410.458,Z 527.077,A -85,B 0,C 180,E1 -10538.865,E2 -10538.865} C_VEL
LIN {X 0,Y 410.698,Z 519.746,A -85,B 0,C 180,E1 -10540.352,E2 -10540.352} C_VEL
LIN {X 0,Y 411.207,Z 510.653,A -85,B 0,C 180,E1 -10541.836,E2 -10541.836} C_VEL
LIN {X 0,Y 411.904,Z 500.716,A -85,B 0,C 180,E1 -10543.144,E2 -10543.144} C_VEL
LIN {X 0,Y 412.517,Z 491.018,A -85,B 0,C 180,E1 -10544.177,E2 -10544.177} C_VEL
LIN {X 0,Y 413.21,Z 479.565,A -85,B 0,C 180,E1 -10545.16,E2 -10545.16} C_VEL
LIN {X 0,Y 413.715,Z 470.73,A -85,B 0,C 180,E1 -10545.772,E2 -10545.772} C_VEL
LIN {X 0,Y 412.779,Z 457.31,A -85,B 0,C 180,E1 -10546.535,E2 -10546.535} C_VEL
LIN {X 0,Y 411.543,Z 444.049,A -85,B 0,C 180,E1 -10547.081,E2 -10547.081} C_VEL
LIN {X 0,Y 410.594,Z 434.582,A -85,B 0,C 180,E1 -10547.379,E2 -10547.379} C_VEL
LIN {X 0,Y 410.968,Z 421.717,A -85,B 0,C 180,E1 -10551.047,E2 -10551.047} C_VEL
LIN {X 0,Y 411.454,Z 409.075,A -85,B 0,C 180,E1 -10554.68,E2 -10554.68} C_VEL
LIN {X 0,Y 412.012,Z 397.746,A -85,B 0,C 180,E1 -10557.975,E2 -10557.975} C_VEL
